			(* Config Cyl ToolTension *)
				ptrTCylToolTension^.T_CtrleCyl.xFBActiv:=TRUE;
				ptrTCylToolTension^.T_Config.xActivState:=TRUE;
				(*22.12.2009: KFS {    *)
				IF xMicroRodActive THEN
				(* Config Cyl ToolLeftActive*)
					ptrTCylToolLeftActive^.T_CtrleCyl.xFBActiv:=TRUE;
					ptrTCylToolLeftActive^.T_Config.xActivState:=TRUE;
				(* Config Cyl ToolRightActive*)
					ptrTCylToolRightActive^.T_CtrleCyl.xFBActiv:=TRUE;
					ptrTCylToolRightActive^.T_Config.xActivState:=TRUE;
				(* Config Cyl ToolCenterActive*)
					ptrTCylToolCenterActive^.T_CtrleCyl.xFBActiv:=TRUE;
					ptrTCylToolCenterActive^.T_Config.xActivState:=TRUE;
				(* Config Cyl ToolPrismaLeftActive*)
					ptrTCylToolPrismaLeftActive^.T_CtrleCyl.xFBActiv:=TRUE;
					ptrTCylToolPrismaLeftActive^.T_Config.xActivState:=TRUE;
				(* Config Cyl ToolPrismaRightActive*)
					ptrTCylToolPrismaRightActive^.T_CtrleCyl.xFBActiv:=TRUE;
					ptrTCylToolPrismaRightActive^.T_Config.xActivState:=TRUE;
				(* Config Cyl ToolWorkLength*)
					ptrTToolFeederWorkLength^.T_CtrleCyl.xFBActiv:=TRUE;
					ptrTToolFeederWorkLength^.T_Config.xActivState:=TRUE;
				END_IF;
				(*22.12.2009: KFS }   *)
			(* Config ToolLeft Axis *)
				ptrTAxisToolLeft^.T_Config_Gen.iTyp:=1;
				ptrTAxisToolLeft^.T_Config_Gen.iMachineType:=iConfigMachineType;
				ptrTAxisToolLeft^.T_Config_ObjFileValue.xSWLimitNeg:=FALSE;
				ptrTAxisToolLeft^.T_Config_ObjFileValue.xSWLimitPos:=FALSE;
				ptrTAxisToolLeft^.T_Config_ObjFileValue.xHWLimitNeg:=FALSE;
				ptrTAxisToolLeft^.T_Config_ObjFileValue.xHWLimitPos:=FALSE;
			(* Config ToolCenter Axis *)
				IF xMicroRodActive THEN
					ptrTAxisToolCenter^.T_Config_Gen.iTyp:=2;
					ptrTAxisToolCenter^.T_Config_Gen.iMachineType:=iConfigMachineType;
					ptrTAxisToolCenter^.T_Config_ObjFileValue.xSWLimitNeg:=FALSE;
					ptrTAxisToolCenter^.T_Config_ObjFileValue.xSWLimitPos:=FALSE;
					ptrTAxisToolCenter^.T_Config_ObjFileValue.xHWLimitNeg:=FALSE;
					ptrTAxisToolCenter^.T_Config_ObjFileValue.xHWLimitPos:=FALSE;
				END_IF;
			(* Config ToolRight Axis *)
				ptrTAxisToolRight^.T_Config_Gen.iTyp:=3;
				ptrTAxisToolRight^.T_Config_Gen.iMachineType:=iConfigMachineType;
				ptrTAxisToolRight^.T_Config_ObjFileValue.xSWLimitNeg:=FALSE;
				ptrTAxisToolRight^.T_Config_ObjFileValue.xSWLimitPos:=FALSE;
				ptrTAxisToolRight^.T_Config_ObjFileValue.xHWLimitNeg:=FALSE;
				ptrTAxisToolRight^.T_Config_ObjFileValue.xHWLimitPos:=FALSE;
			(* Config ToolFeeder Axis *)
				ptrTAxisToolFeeder^.T_Config_Gen.iTyp:=4;
				ptrTAxisToolFeeder^.T_Config_Gen.iMachineType:=iConfigMachineType;
				IF xMicroRodActive THEN
					ptrTAxisToolFeeder^.T_Config_ObjFileValue.xSWLimitNeg:=FALSE;
					ptrTAxisToolFeeder^.T_Config_ObjFileValue.xSWLimitPos:=FALSE;
				   	ptrTAxisToolFeeder^.T_Config_ObjFileValue.xHWLimitNeg:=TRUE;
					ptrTAxisToolFeeder^.T_Config_ObjFileValue.xHWLimitPos:=TRUE;
				ELSE
					ptrTAxisToolFeeder^.T_Config_ObjFileValue.xSWLimitNeg:=FALSE;
					ptrTAxisToolFeeder^.T_Config_ObjFileValue.xSWLimitPos:=FALSE;
					ptrTAxisToolFeeder^.T_Config_ObjFileValue.xHWLimitNeg:=FALSE;
					ptrTAxisToolFeeder^.T_Config_ObjFileValue.xHWLimitPos:=FALSE;
				END_IF;
			(* Config GrindFeeder Axis *)
				ptrTAxisGrindFeeder^.T_Config_Gen.iTyp:=5;
				ptrTAxisGrindFeeder^.T_Config_Gen.iMachineType:=iConfigMachineType;
				ptrTAxisGrindFeeder^.T_Config_ObjFileValue.xSWLimitNeg:=TRUE;
				ptrTAxisGrindFeeder^.T_Config_ObjFileValue.xSWLimitPos:=TRUE;
				ptrTAxisGrindFeeder^.T_Config_ObjFileValue.xHWLimitNeg:=FALSE;
				ptrTAxisGrindFeeder^.T_Config_ObjFileValue.xHWLimitPos:=FALSE;
			END_IF;
			IF NOT(ptrTFunction^.xReset) AND ptrTFunction^.xEnd THEN
				(* Alle Funktionen Resetten *)
				IF (iStationFunctionNr < iMaxFunctionNr) THEN
					iStationFunctionNr:=iStationFunctionNr + 1;
					ptrTFunction^.xReset:=TRUE;
				ELSE
					xInitStep:=FALSE;
					xStartFunction:=FALSE;
					iStepEnable:=200;
				END_IF;
			END_IF;
		110:	IF NOT(xInitStep) THEN
				xInitStep:=TRUE;
				IF TStation.TControl.xHardwareConfigError THEN
					TStation.TControl.xHardwareConfigError:=FALSE;
					TStation.TControl.xActiveHardware:=FALSE;
				ELSE
					xRdyDisableStation:=TRUE;
					xInitStep:=FALSE;
					iStepEnable:=100;
				END_IF;
				RETURN;
			END_IF;
			IF NOT(TStation.TControl.xError) THEN
				TStation.TControl.xActiveHardware:=TRUE;
				xRdyDisableStation:=TRUE;
				xInitStep:=FALSE;
				iStepEnable:=100;
				RETURN;
			END_IF;
		200:	IF NOT(xInitStep) THEN
				xInitStep:=TRUE;
				ptrTCylToolTension^.T_CtrleCyl.xReset:=TRUE;
				(*22.12.2009: KFS {    *)
				IF xMicroRodActive THEN
					ptrTCylToolLeftActive^.T_CtrleCyl.xReset:=TRUE;
					ptrTCylToolRightActive^.T_CtrleCyl.xReset:=TRUE;
					ptrTCylToolCenterActive^.T_CtrleCyl.xReset:=TRUE;
					ptrTCylToolPrismaLeftActive^.T_CtrleCyl.xReset:=TRUE;
					ptrTCylToolPrismaRightActive^.T_CtrleCyl.xReset:=TRUE;
					ptrTToolFeederWorkLength^.T_CtrleCyl.xReset:=TRUE;
				END_IF;
				(*22.12.2009: KFS }   *)
				ptrTAxisToolLeft^.T_CtrleSingle.xReset:=TRUE;
				IF xMicroRodActive THEN
					ptrTAxisToolCenter^.T_CtrleSingle.xReset:=TRUE;
				END_IF;
				ptrTAxisToolRight^.T_CtrleSingle.xReset:=TRUE;
				ptrTAxisToolFeeder^.T_CtrleSingle.xReset:=TRUE;
				ptrTAxisGrindFeeder^.T_CtrleSingle.xReset:=TRUE;
				ptrTAxisGrindSpindle^.T_CtrleSingle.xReset:=TRUE;
			END_IF;
			IF NOT(ptrTAxisToolLeft^.T_CtrleSingle.xReset) AND NOT(ptrTAxisToolCenter^.T_CtrleSingle.xReset) AND ((NOT(ptrTAxisToolRight^.T_CtrleSingle.xReset) AND xMicroRodActive) OR NOT(xMicroRodActive)) AND
			     NOT(ptrTAxisToolFeeder^.T_CtrleSingle.xReset) AND NOT(ptrTAxisGrindFeeder^.T_CtrleSingle.xReset) AND NOT(ptrTAxisGrindSpindle^.T_CtrleSingle.xReset) THEN
				xInitStep:=FALSE;
				IF NOT(xBeckhoffDriveActive) THEN
					iStepEnable:=300;
				ELSE
					iStepEnable:=500;
				END_IF;
			END_IF;
		300:	IF NOT(xInitStep) THEN
				xInitStep:=TRUE;
				ptrTAxisToolLeft^.T_CtrleSingle.lrAcceleration:=T_Standard.T_TeachINToolLeft.rAcceleration;
				ptrTAxisToolLeft^.T_CtrleSingle.lrDecceleration:=T_Standard.T_TeachINToolLeft.rDeceleration;
				ptrTAxisToolCenter^.T_CtrleSingle.lrAcceleration:=T_Standard.T_TeachINToolCenter.rAcceleration;
				ptrTAxisToolCenter^.T_CtrleSingle.lrDecceleration:=T_Standard.T_TeachINToolCenter.rDeceleration;
				ptrTAxisToolRight^.T_CtrleSingle.lrAcceleration:=T_Standard.T_TeachINToolRight.rAcceleration;
				ptrTAxisToolRight^.T_CtrleSingle.lrDecceleration:=T_Standard.T_TeachINToolRight.rDeceleration;
				ptrTAxisToolFeeder^.T_CtrleSingle.lrAcceleration:=T_Standard.T_TeachINToolFeeder.rAcceleration;
				ptrTAxisToolFeeder^.T_CtrleSingle.lrDecceleration:=T_Standard.T_TeachINToolFeeder.rDeceleration;
				ptrTAxisGrindFeeder^.T_CtrleSingle.lrAcceleration:=T_Standard.T_TeachINGrindFeeder.rAcceleration;
				ptrTAxisGrindFeeder^.T_CtrleSingle.lrDecceleration:=T_Standard.T_TeachINGrindFeeder.rDeceleration;
				ptrTAxisToolLeft^.T_Config_Gen.sFileNamePDOMapping:='PDOMapping_ToolLeft';
				ptrTAxisToolLeft^.T_CtrleSingle.iFunction:=22;
				ptrTAxisToolLeft^.T_CtrleSingle.xExecute:=TRUE;
				IF xMicroRodActive THEN
					ptrTAxisToolCenter^.T_Config_Gen.sFileNamePDOMapping:='PDOMapping_ToolCenter';
					ptrTAxisToolCenter^.T_CtrleSingle.iFunction:=22;
					ptrTAxisToolCenter^.T_CtrleSingle.xExecute:=TRUE;
				END_IF;
				ptrTAxisToolRight^.T_Config_Gen.sFileNamePDOMapping:='PDOMapping_ToolRight';
				ptrTAxisToolRight^.T_CtrleSingle.iFunction:=22;
				ptrTAxisToolRight^.T_CtrleSingle.xExecute:=TRUE;
				ptrTAxisToolFeeder^.T_Config_Gen.sFileNamePDOMapping:='PDOMapping_ToolFeeder';
				ptrTAxisToolFeeder^.T_CtrleSingle.iFunction:=22;
				ptrTAxisToolFeeder^.T_CtrleSingle.xExecute:=TRUE;
				ptrTAxisGrindFeeder^.T_Config_Gen.sFileNamePDOMapping:='PDOMapping_GrindFeeder';
				ptrTAxisGrindFeeder^.T_CtrleSingle.iFunction:=22;
				ptrTAxisGrindFeeder^.T_CtrleSingle.xExecute:=TRUE;
				iCountCycle:=0;
			END_IF;
			iCountCycle:=iCountCycle + 1;
			IF (iCountCycle >= 50) THEN
				xReadyChkError:=TRUE;	(* 50 SPS Zyklen warten bis die Übewachung der HW Error freigeschaltet werden kann *)
			END_IF;
			IF xTmp THEN
				RETURN;	(* Wait until all Drives finished *)
			END_IF;
			IF NOT(ptrTAxisToolLeft^.T_CtrleSingle.xExecute) AND ptrTAxisToolLeft^.T_CtrleSingle.xDone AND
			    ((NOT(ptrTAxisToolCenter^.T_CtrleSingle.xExecute) AND ptrTAxisToolCenter^.T_CtrleSingle.xDone AND xMicroRodActive) OR NOT(xMicroRodActive)) AND
			    NOT(ptrTAxisToolRight^.T_CtrleSingle.xExecute) AND ptrTAxisToolRight^.T_CtrleSingle.xDone AND
			    NOT(ptrTAxisToolFeeder^.T_CtrleSingle.xExecute) AND ptrTAxisToolFeeder^.T_CtrleSingle.xDone AND
			    NOT(ptrTAxisGrindFeeder^.T_CtrleSingle.xExecute) AND ptrTAxisGrindFeeder^.T_CtrleSingle.xDone THEN
				xReadyChkError:=TRUE;
				xInitStep:=FALSE;
				iStepEnable:=400;
			END_IF;
		400:	IF NOT(xInitStep) THEN
				xInitStep:=TRUE;
				ptrTAxisToolLeft^.T_CtrleSingle.iFunction:=23;
				ptrTAxisToolLeft^.T_CtrleSingle.xExecute:=TRUE;
				IF xMicroRodActive THEN
					ptrTAxisToolCenter^.T_CtrleSingle.iFunction:=23;
					ptrTAxisToolCenter^.T_CtrleSingle.xExecute:=TRUE;
				END_IF;
				ptrTAxisToolRight^.T_CtrleSingle.iFunction:=23;
				ptrTAxisToolRight^.T_CtrleSingle.xExecute:=TRUE;
				ptrTAxisToolFeeder^.T_CtrleSingle.iFunction:=23;
				ptrTAxisToolFeeder^.T_CtrleSingle.xExecute:=TRUE;
				ptrTAxisGrindFeeder^.T_CtrleSingle.iFunction:=23;
				ptrTAxisGrindFeeder^.T_CtrleSingle.xExecute:=TRUE;
			END_IF;
			IF xTmp THEN
				RETURN;	(* Wait until all Drives finished *)
			END_IF;
			IF NOT(ptrTAxisToolLeft^.T_CtrleSingle.xExecute) AND ptrTAxisToolLeft^.T_CtrleSingle.xDone AND
			    ((NOT(ptrTAxisToolCenter^.T_CtrleSingle.xExecute) AND ptrTAxisToolCenter^.T_CtrleSingle.xDone AND xMicroRodActive) OR NOT(xMicroRodActive)) AND
			    NOT(ptrTAxisToolRight^.T_CtrleSingle.xExecute) AND ptrTAxisToolRight^.T_CtrleSingle.xDone AND
			    NOT(ptrTAxisToolFeeder^.T_CtrleSingle.xExecute) AND ptrTAxisToolFeeder^.T_CtrleSingle.xDone AND
			    NOT(ptrTAxisGrindFeeder^.T_CtrleSingle.xExecute) AND ptrTAxisGrindFeeder^.T_CtrleSingle.xDone THEN
				xInitStep:=FALSE;
				iStepEnable:=500;
			END_IF;
		500:	IF NOT(xInitStep) THEN
				xInitStep:=TRUE;
				ptrTAxisToolLeft^.T_CtrleSingle.iFunction:=1;
				ptrTAxisToolLeft^.T_CtrleSingle.xExecute:=TRUE;
				IF xMicroRodActive THEN
					ptrTAxisToolCenter^.T_CtrleSingle.iFunction:=1;
					ptrTAxisToolCenter^.T_CtrleSingle.xExecute:=TRUE;
				END_IF;
				ptrTAxisToolRight^.T_CtrleSingle.iFunction:=1;
				ptrTAxisToolRight^.T_CtrleSingle.xExecute:=TRUE;
				ptrTAxisToolFeeder^.T_CtrleSingle.iFunction:=1;
				ptrTAxisToolFeeder^.T_CtrleSingle.xExecute:=TRUE;
				ptrTAxisGrindFeeder^.T_CtrleSingle.iFunction:=1;
				ptrTAxisGrindFeeder^.T_CtrleSingle.xExecute:=TRUE;
			END_IF;
			IF NOT(ptrTAxisToolLeft^.T_CtrleSingle.xExecute) AND ptrTAxisToolLeft^.T_CtrleSingle.xDone AND
			    ((NOT(ptrTAxisToolCenter^.T_CtrleSingle.xExecute) AND ptrTAxisToolCenter^.T_CtrleSingle.xDone AND xMicroRodActive) OR NOT(xMicroRodActive)) AND
			    NOT(ptrTAxisToolRight^.T_CtrleSingle.xExecute) AND ptrTAxisToolRight^.T_CtrleSingle.xDone AND
			    NOT(ptrTAxisToolFeeder^.T_CtrleSingle.xExecute) AND ptrTAxisToolFeeder^.T_CtrleSingle.xDone AND
			    NOT(ptrTAxisGrindFeeder^.T_CtrleSingle.xExecute) AND ptrTAxisGrindFeeder^.T_CtrleSingle.xDone THEN
				xInitStep:=FALSE;
				iStepEnable:=600;
			END_IF;
		600:	IF NOT(xInitStep) THEN	(* Read Axis Parameter File *)
				xInitStep:=TRUE;
				ptrTAxisToolLeft^.T_Config_Gen.sDeviceFileName:='EcoStep23S21_ToolLeft';
				ptrTAxisToolLeft^.T_CtrleSingle.iFunction:=2;
				ptrTAxisToolLeft^.T_CtrleSingle.xExecute:=TRUE;
				IF xMicroRodActive THEN
					ptrTAxisToolCenter^.T_Config_Gen.sDeviceFileName:='EcoStep23S21_ToolCenter';
					ptrTAxisToolCenter^.T_CtrleSingle.iFunction:=2;
					ptrTAxisToolCenter^.T_CtrleSingle.xExecute:=TRUE;
				END_IF;
				ptrTAxisToolRight^.T_Config_Gen.sDeviceFileName:='EcoStep23S21_ToolRight';
				ptrTAxisToolRight^.T_CtrleSingle.iFunction:=2;
				ptrTAxisToolRight^.T_CtrleSingle.xExecute:=TRUE;
				ptrTAxisToolFeeder^.T_Config_Gen.sDeviceFileName:='EcoStep23S21_ToolFeeder';
				ptrTAxisToolFeeder^.T_CtrleSingle.iFunction:=2;
				ptrTAxisToolFeeder^.T_CtrleSingle.xExecute:=TRUE;
				ptrTAxisGrindFeeder^.T_Config_Gen.sDeviceFileName:='EcoStep23S21_GrindFeeder';
				ptrTAxisGrindFeeder^.T_CtrleSingle.iFunction:=2;
				ptrTAxisGrindFeeder^.T_CtrleSingle.xExecute:=TRUE;
			END_IF;
			IF NOT(ptrTAxisToolLeft^.T_CtrleSingle.xExecute) AND ptrTAxisToolLeft^.T_CtrleSingle.xDone AND
			    ((NOT(ptrTAxisToolCenter^.T_CtrleSingle.xExecute) AND ptrTAxisToolCenter^.T_CtrleSingle.xDone AND xMicroRodActive) OR NOT(xMicroRodActive)) AND
			    NOT(ptrTAxisToolRight^.T_CtrleSingle.xExecute) AND ptrTAxisToolRight^.T_CtrleSingle.xDone AND
			    NOT(ptrTAxisToolFeeder^.T_CtrleSingle.xExecute) AND ptrTAxisToolFeeder^.T_CtrleSingle.xDone AND
			    NOT(ptrTAxisGrindFeeder^.T_CtrleSingle.xExecute) AND ptrTAxisGrindFeeder^.T_CtrleSingle.xDone THEN
				xInitStep:=FALSE;
				iStepEnable:=700;
			END_IF;
		700:	IF NOT(xInitStep) THEN	(* Read Axis Parameter File *)
				xInitStep:=TRUE;
				ptrTAxisToolLeft^.T_CtrleSingle.iFunction:=21;
				ptrTAxisToolLeft^.T_CtrleSingle.xExecute:=TRUE;
				IF xMicroRodActive THEN
					ptrTAxisToolCenter^.T_CtrleSingle.iFunction:=21;
					ptrTAxisToolCenter^.T_CtrleSingle.xExecute:=TRUE;
				END_IF;
				ptrTAxisToolRight^.T_CtrleSingle.iFunction:=21;
				ptrTAxisToolRight^.T_CtrleSingle.xExecute:=TRUE;
				ptrTAxisToolFeeder^.T_CtrleSingle.iFunction:=21;
				ptrTAxisToolFeeder^.T_CtrleSingle.xExecute:=TRUE;
				ptrTAxisGrindFeeder^.T_CtrleSingle.iFunction:=21;
				ptrTAxisGrindFeeder^.T_CtrleSingle.xExecute:=TRUE;
			END_IF;
			IF NOT(ptrTAxisToolLeft^.T_CtrleSingle.xExecute) AND ptrTAxisToolLeft^.T_CtrleSingle.xDone AND
			    ((NOT(ptrTAxisToolCenter^.T_CtrleSingle.xExecute) AND ptrTAxisToolCenter^.T_CtrleSingle.xDone AND xMicroRodActive) OR NOT(xMicroRodActive)) AND
			    NOT(ptrTAxisToolRight^.T_CtrleSingle.xExecute) AND ptrTAxisToolRight^.T_CtrleSingle.xDone AND
			    NOT(ptrTAxisToolFeeder^.T_CtrleSingle.xExecute) AND ptrTAxisToolFeeder^.T_CtrleSingle.xDone AND
			    NOT(ptrTAxisGrindFeeder^.T_CtrleSingle.xExecute) AND ptrTAxisGrindFeeder^.T_CtrleSingle.xDone THEN
				xInitStep:=FALSE;
				IF NOT(xBeckhoffDriveActive) THEN
					iStepEnable:=1000;
				ELSE
					iStepEnable:=800;
				END_IF;
			END_IF;
		800:	IF NOT(xInitStep) THEN
				IF NOT(T_BoxID.T_Ctrle.xLocked) THEN
					xInitStep:=TRUE;
					(* Box ID-->Beckhoff drive *)
					T_BoxID.T_Ctrle.iMachineType:=iConfigMachineType;
					T_BoxID.T_Servo_ToolLeft.sBoxName:='AX25xx_Slide_St1';
					T_BoxID.T_Servo_ToolLeft.sDeviceName:='AX25xx_Slide_St1';
					T_BoxID.T_Servo_ToolLeft.xDeviceOption:=TRUE;
					T_BoxID.T_Servo_ToolCenter.sBoxName:='AX25xx_Slide_St1';
					T_BoxID.T_Servo_ToolCenter.sDeviceName:='AX25xx_Slide_St1';
					T_BoxID.T_Servo_ToolCenter.xDeviceOption:=TRUE;
					T_BoxID.T_Servo_ToolRight.sBoxName:='AX25xx_Slide_St1';
					T_BoxID.T_Servo_ToolRight.sDeviceName:='AX25xx_Slide_St1';
					T_BoxID.T_Servo_ToolRight.xDeviceOption:=TRUE;
					T_BoxID.T_Servo_ToolFeeder.sBoxName:='AX25xx_Slide_St1';
					T_BoxID.T_Servo_ToolFeeder.sDeviceName:='AX25xx_Slide_St1';
					T_BoxID.T_Servo_ToolFeeder.xDeviceOption:=TRUE;
					T_BoxID.T_Servo_GrindFeeder.sBoxName:='AX25xx_Slide_St1';
					T_BoxID.T_Servo_GrindFeeder.sDeviceName:='AX25xx_Slide_St1';
					T_BoxID.T_Servo_GrindFeeder.xDeviceOption:=TRUE;
					T_BoxID.T_Ctrle.xLocked:=TRUE;
					T_BoxID.T_Ctrle.xExecute:=TRUE;
				END_IF;
				RETURN;
			END_IF;
			IF NOT(T_BoxID.T_Ctrle.xExecute) AND T_BoxID.T_Ctrle.xDone AND T_BoxID.T_Ctrle.xLocked THEN
				T_BoxID.T_Ctrle.xLocked:=FALSE;
				xInitStep:=FALSE;
				iStepEnable:=900;
			END_IF;
		900:	IF NOT(xInitStep) THEN
				xInitStep:=TRUE;
				IF (T_BoxID.T_Servo_ToolLeft.wAddrBox = 0) OR (T_BoxID.T_Servo_ToolLeft.wAddrBox <> ptrTAxisToolLeft^.T_Config_Gen.udiNC_TaskIdxGrp) THEN
					xSetError:=TRUE;
					diErrorNumber:=16#F201;	(* ToolLeft-->Falsche Konfiguration oder Achse nicht vorhanden *)
					RETURN;
				ELSIF ((T_BoxID.T_Servo_ToolCenter.wAddrBox = 0) OR (T_BoxID.T_Servo_ToolCenter.wAddrBox <> ptrTAxisToolCenter^.T_Config_Gen.udiNC_TaskIdxGrp)) AND xMicroRodActive THEN
					xSetError:=TRUE;
					diErrorNumber:=16#F202;	(* ToolCenter-->Falsche Konfiguration oder Achse nicht vorhanden *)
					RETURN;
				ELSIF (T_BoxID.T_Servo_ToolRight.wAddrBox = 0) OR (T_BoxID.T_Servo_ToolRight.wAddrBox <> ptrTAxisToolRight^.T_Config_Gen.udiNC_TaskIdxGrp) THEN
					xSetError:=TRUE;
					diErrorNumber:=16#F203;	(* ToolRight-->Falsche Konfiguration oder Achse nicht vorhanden *)
					RETURN;
				ELSIF (T_BoxID.T_Servo_ToolFeeder.wAddrBox = 0) OR (T_BoxID.T_Servo_ToolFeeder.wAddrBox <> ptrTAxisToolFeeder^.T_Config_Gen.udiNC_TaskIdxGrp) THEN
					xSetError:=TRUE;
					diErrorNumber:=16#F204;	(* ToolFeeder-->Falsche Konfiguration oder Achse nicht vorhanden *)
					RETURN;
				ELSIF (T_BoxID.T_Servo_GrindFeeder.wAddrBox = 0) OR (T_BoxID.T_Servo_GrindFeeder.wAddrBox <> ptrTAxisGrindFeeder^.T_Config_Gen.udiNC_TaskIdxGrp) THEN
					xSetError:=TRUE;
					diErrorNumber:=16#F205;	(* GrindFeeder-->Falsche Konfiguration oder Achse nicht vorhanden *)
					RETURN;
				ELSE
				(* Achsenparameterisierung erfolgreich *)
					;
				END_IF;
				xInitStep:=FALSE;
				iStepEnable:=1100;
			END_IF;
		(* Read Axis Firmware Information *)
		1000:IF NOT(xInitStep) THEN
				xInitStep:=TRUE;
				ptrTAxisToolLeft^.T_CtrleSingle.iFunction:=27;
				ptrTAxisToolLeft^.T_CtrleSingle.xExecute:=TRUE;
				IF xMicroRodActive THEN
					ptrTAxisToolCenter^.T_CtrleSingle.iFunction:=27;
					ptrTAxisToolCenter^.T_CtrleSingle.xExecute:=TRUE;
				END_IF;
				ptrTAxisToolRight^.T_CtrleSingle.iFunction:=27;
				ptrTAxisToolRight^.T_CtrleSingle.xExecute:=TRUE;
				ptrTAxisToolFeeder^.T_CtrleSingle.iFunction:=27;
				ptrTAxisToolFeeder^.T_CtrleSingle.xExecute:=TRUE;
				ptrTAxisGrindFeeder^.T_CtrleSingle.iFunction:=27;
				ptrTAxisGrindFeeder^.T_CtrleSingle.xExecute:=TRUE;
			END_IF;
			IF NOT(ptrTAxisToolLeft^.T_CtrleSingle.xExecute) AND ptrTAxisToolLeft^.T_CtrleSingle.xDone AND
			    ((NOT(ptrTAxisToolCenter^.T_CtrleSingle.xExecute) AND ptrTAxisToolCenter^.T_CtrleSingle.xDone AND xMicroRodActive) OR NOT(xMicroRodActive)) AND
			    NOT(ptrTAxisToolRight^.T_CtrleSingle.xExecute) AND ptrTAxisToolRight^.T_CtrleSingle.xDone AND
			    NOT(ptrTAxisToolFeeder^.T_CtrleSingle.xExecute) AND ptrTAxisToolFeeder^.T_CtrleSingle.xDone AND
			    NOT(ptrTAxisGrindFeeder^.T_CtrleSingle.xExecute) AND ptrTAxisGrindFeeder^.T_CtrleSingle.xDone THEN
				xInitStep:=FALSE;
				iStepEnable:=1100;
			END_IF;
		1100:IF NOT(xInitStep) THEN
				xInitStep:=TRUE;
				ptrTAxisToolLeft^.T_CtrleSingle.iFunction:=4;
				ptrTAxisToolLeft^.T_CtrleSingle.xExecute:=TRUE;
				IF xMicroRodActive THEN
					ptrTAxisToolCenter^.T_CtrleSingle.iFunction:=4;
					ptrTAxisToolCenter^.T_CtrleSingle.xExecute:=TRUE;
				END_IF;
				ptrTAxisToolRight^.T_CtrleSingle.iFunction:=4;
				ptrTAxisToolRight^.T_CtrleSingle.xExecute:=TRUE;
				ptrTAxisToolFeeder^.T_CtrleSingle.iFunction:=4;
				ptrTAxisToolFeeder^.T_CtrleSingle.xExecute:=TRUE;
				ptrTAxisGrindFeeder^.T_CtrleSingle.iFunction:=4;
				ptrTAxisGrindFeeder^.T_CtrleSingle.xExecute:=TRUE;
				ptrTAxisGrindSpindle^.T_CtrleSingle.iFunction:=4;
				ptrTAxisGrindSpindle^.T_CtrleSingle.xExecute:=TRUE;
			END_IF;
			IF NOT(ptrTAxisToolLeft^.T_CtrleSingle.xExecute) AND ptrTAxisToolLeft^.T_CtrleSingle.xDone AND
			    ((NOT(ptrTAxisToolCenter^.T_CtrleSingle.xExecute) AND ptrTAxisToolCenter^.T_CtrleSingle.xDone AND xMicroRodActive) OR NOT(xMicroRodActive)) AND
			    NOT(ptrTAxisToolRight^.T_CtrleSingle.xExecute) AND ptrTAxisToolRight^.T_CtrleSingle.xDone AND
			    NOT(ptrTAxisToolFeeder^.T_CtrleSingle.xExecute) AND ptrTAxisToolFeeder^.T_CtrleSingle.xDone AND
			    NOT(ptrTAxisGrindFeeder^.T_CtrleSingle.xExecute) AND ptrTAxisGrindFeeder^.T_CtrleSingle.xDone AND
			    NOT(ptrTAxisGrindSpindle^.T_CtrleSingle.xExecute) AND ptrTAxisGrindSpindle^.T_CtrleSingle.xDone THEN
				xInitStep:=FALSE;
				iStepEnable:=1200;
			END_IF;
		1200:IF NOT(xInitStep) THEN
				xInitStep:=TRUE;
				ptrTAxisToolLeft^.T_CtrleSingle.iFunction:=3;
				ptrTAxisToolLeft^.T_CtrleSingle.xExecute:=TRUE;
				IF xMicroRodActive THEN
					ptrTAxisToolCenter^.T_CtrleSingle.iFunction:=3;
					ptrTAxisToolCenter^.T_CtrleSingle.xExecute:=TRUE;
				END_IF;
				ptrTAxisToolRight^.T_CtrleSingle.iFunction:=3;
				ptrTAxisToolRight^.T_CtrleSingle.xExecute:=TRUE;
				ptrTAxisToolFeeder^.T_CtrleSingle.iFunction:=3;
				ptrTAxisToolFeeder^.T_CtrleSingle.xExecute:=TRUE;
				ptrTAxisGrindFeeder^.T_CtrleSingle.iFunction:=3;
				ptrTAxisGrindFeeder^.T_CtrleSingle.xExecute:=TRUE;
			END_IF;
			IF NOT(ptrTAxisToolLeft^.T_CtrleSingle.xExecute) AND ptrTAxisToolLeft^.T_CtrleSingle.xDone AND
			    ((NOT(ptrTAxisToolCenter^.T_CtrleSingle.xExecute) AND ptrTAxisToolCenter^.T_CtrleSingle.xDone AND xMicroRodActive) OR NOT(xMicroRodActive)) AND
			    NOT(ptrTAxisToolRight^.T_CtrleSingle.xExecute) AND ptrTAxisToolRight^.T_CtrleSingle.xDone AND
			    NOT(ptrTAxisToolFeeder^.T_CtrleSingle.xExecute) AND ptrTAxisToolFeeder^.T_CtrleSingle.xDone AND
			    NOT(ptrTAxisGrindFeeder^.T_CtrleSingle.xExecute) AND ptrTAxisGrindFeeder^.T_CtrleSingle.xDone THEN
				IF NOT(xFirstTimeBooting) THEN
					xFirstTimeBooting:=TRUE;
					iStepEnable:=1300;
				ELSE
					iStepEnable:=1400;
				END_IF;
				xInitStep:=FALSE;
			END_IF;
		(* Set the Position of the GrindFeeder on the Settled ToolDiameter, but only on the first time on booting of the machine *)
		1300:IF NOT(xInitStep) THEN
				xInitStep:=TRUE;
				ptrTAxisGrindFeeder^.T_CtrleSingle.rSetPosition:=T_ProcessImageData.T_ProcessPara.rToolDiameterProcess;
				ptrTAxisGrindFeeder^.T_CtrleSingle.iFunction:=11;
				ptrTAxisGrindFeeder^.T_CtrleSingle.xExecute:=TRUE;
			END_IF;
			IF NOT(ptrTAxisGrindFeeder^.T_CtrleSingle.xExecute) AND ptrTAxisGrindFeeder^.T_CtrleSingle.xDone THEN
				xInitStep:=FALSE;
				iStepEnable:=1400;
			END_IF;
		(* Set the SW Limit position for the GrindFeeder Axis *)
		1400:IF NOT(xInitStep) THEN
				xInitStep:=TRUE;
				ptrTAxisGrindFeeder^.T_CtrleSingle.lrSWNegLimitSwitch:=T_ProcessImageData.T_PrismPara.rToolDiameterMin;
				ptrTAxisGrindFeeder^.T_CtrleSingle.lrSWPosLimitSwitch:=T_ProcessImageData.T_PrismPara.rToolDiameterMax + T_Standard.T_TeachINGrindFeeder.rOffsetSWPosEndSwitch;
				ptrTAxisGrindFeeder^.T_CtrleSingle.iFunction:=28;
				ptrTAxisGrindFeeder^.T_CtrleSingle.xExecute:=TRUE;
			END_IF;
			IF NOT(ptrTAxisGrindFeeder^.T_CtrleSingle.xExecute) AND ptrTAxisGrindFeeder^.T_CtrleSingle.xDone THEN
				xInitStep:=FALSE;
				IF NOT(xMicroRodActive) THEN
					(* Only for MicroWire activate the ToolTension *)
					iStepEnable:=1500;
				ELSE
					iStepEnable:=1600;
				END_IF;
			END_IF;
		1500:IF NOT(xInitStep) THEN
				xInitStep:=TRUE;
				ptrTCylToolTension^.T_CtrleCyl.iFunction:=2;
				ptrTCylToolTension^.T_CtrleCyl.T_AnalogCylinder.rForceIn:=T_ProcessImageData.T_ProcessPara.rToolTensionProcess;
				ptrTCylToolTension^.T_CtrleCyl.xExecute:=TRUE;
			END_IF;
			IF NOT(ptrTCylToolTension^.T_CtrleCyl.xExecute) AND ptrTCylToolTension^.T_CtrleCyl.xDone THEN
				xInitStep:=FALSE;
				iStepEnable:=1600;
			END_IF;
		1600:xReadyChkError:=FALSE;
			xInitStep:=FALSE;
			xSetEnableConfig:=TRUE;
			iEnableConfigMachineType:=iConfigMachineType;
			iEnableConfigAxisType:=iConfigAxisType;
			iEnableConfigVisuNavigation:=iConfigVisuNavigation;
			rEnableConfigMaxToolLength:=rConfigMaxToolLength;
			xInitSetEnable:=FALSE;
			TStation.TControl.xRdy:=TRUE;
			xSetEnd:=TRUE;
	END_CASE;
END_IF;
END_ACTION
ACTION CtrlErrorStation:
IF xStationError OR xForceHWError OR (ptrTFunction^.xError AND TStation.TControl.xRdy AND NOT(xSetEnd)) THEN
	IF NOT(xInitError) THEN
		xForceHWError:=FALSE;
		xStationError:=TRUE;
		xTmpStationError:=TRUE;
		xInitError:=TRUE;
		xAxisErrorActive:=FALSE;
		TStation.TControl.diErrorNr:=0;
		IF ptrTAxisToolLeft^.T_CtrleSingle.xErr THEN
			TStation.TControl.diErrorNr:=1000000 + ptrTAxisToolLeft^.T_CtrleSingle.udiErrorID;
			ptrTAxisToolLeft^.T_CtrleSingle.iFunction:=1;
			ptrTAxisToolLeft^.T_CtrleSingle.xExecute:=TRUE;
			xAxisErrorActive:=TRUE;
		END_IF;
		IF xMicroRodActive THEN
			IF ptrTAxisToolCenter^.T_CtrleSingle.xErr THEN
				TStation.TControl.diErrorNr:=2000000 + ptrTAxisToolCenter^.T_CtrleSingle.udiErrorID;
				ptrTAxisToolCenter^.T_CtrleSingle.iFunction:=1;
				ptrTAxisToolCenter^.T_CtrleSingle.xExecute:=TRUE;
				xAxisErrorActive:=TRUE;
			END_IF;
		END_IF;
		IF ptrTAxisToolRight^.T_CtrleSingle.xErr THEN
			TStation.TControl.diErrorNr:=3000000 + ptrTAxisToolRight^.T_CtrleSingle.udiErrorID;
			ptrTAxisToolRight^.T_CtrleSingle.iFunction:=1;
			ptrTAxisToolRight^.T_CtrleSingle.xExecute:=TRUE;
			xAxisErrorActive:=TRUE;
		END_IF;
		IF ptrTAxisToolFeeder^.T_CtrleSingle.xErr THEN
			TStation.TControl.diErrorNr:=4000000 + ptrTAxisToolFeeder^.T_CtrleSingle.udiErrorID;
			ptrTAxisToolFeeder^.T_CtrleSingle.iFunction:=1;
			ptrTAxisToolFeeder^.T_CtrleSingle.xExecute:=TRUE;
			xAxisErrorActive:=TRUE;
		END_IF;
		IF ptrTAxisGrindFeeder^.T_CtrleSingle.xErr THEN
			TStation.TControl.diErrorNr:=5000000 + ptrTAxisGrindFeeder^.T_CtrleSingle.udiErrorID;
			ptrTAxisGrindFeeder^.T_CtrleSingle.iFunction:=1;
			ptrTAxisGrindFeeder^.T_CtrleSingle.xExecute:=TRUE;
			xAxisErrorActive:=TRUE;
		END_IF;
		IF ptrTCylToolTension^.T_CtrleCyl.xErr THEN
			TStation.TControl.diErrorNr:=6000000 + ptrTCylToolTension^.T_CtrleCyl.udiErrorID;
			ptrTCylToolTension^.T_CtrleCyl.xReset:=TRUE;
		END_IF;
		IF (TStation.TControl.diErrorNr = 0) THEN	(* General Error-->No Hardware Error  7000 - 7999*)
			TStation.TControl.diErrorNr:=8000000 + ptrTFunction^.iErrorNr;
		END_IF;
		ptrTFunction^.xQuitErr:=NOT(ptrTFunction^.xEnd) AND ptrTFunction^.xError;
		IF NOT(ptrTFunction^.xQuitErr) AND NOT(ptrTFunction^.xEnd) THEN
			xForceResetAxis:=TRUE;
			ptrTFunction^.xReset:=TRUE;
		END_IF;
		TONWaitReset(IN:=FALSE);
	END_IF;
	IF (ptrTFunction^.xEnd OR xForceResetAxis) AND xTmpStationError THEN
		IF NOT(ptrTAxisToolLeft^.T_CtrleSingle.xErr) AND ((NOT(ptrTAxisToolCenter^.T_CtrleSingle.xErr) AND xMicroRodActive) OR NOT(xMicroRodActive)) AND
		     NOT(ptrTAxisToolRight^.T_CtrleSingle.xErr) AND NOT(ptrTAxisToolFeeder^.T_CtrleSingle.xErr) AND NOT(ptrTAxisGrindFeeder^.T_CtrleSingle.xErr) THEN
			TStation.TControl.xError:=TRUE;
			xForceResetAxis:=FALSE;
		END_IF;
		TONWaitReset(IN:=TRUE,PT:=T#100ms);
		IF TONWaitReset.Q THEN
			IF xAxisErrorActive THEN
				T_StartUp.T_Ctrle.xSetSecurityStateON:=TRUE;
			END_IF;
			xStepError:=FALSE;
			xStartFunction:=FALSE;
			xTmpStationError:=FALSE;
			xReadyToQuitErr:=TRUE;
		END_IF;
	END_IF;
	IF TStation.TControl.xQuitError AND NOT(ptrTFunction^.xQuitErr) AND xReadyToQuitErr THEN
		xInitError:=FALSE;
		TStation.TControl.xQuitError:=FALSE;
		xSetEnd:=TRUE;
	END_IF;
END_IF;
END_ACTION
ACTION CtrlMainStation:
IF (TStation.TControl.xStart OR xTmpStart) AND TStation.TControl.xRdy AND NOT(xSetEnd) THEN
	IF NOT(xInitStart) THEN
		xInitStart:=TRUE;
		xTmpStart:=TRUE;
		TStation.TControl.xStart:=FALSE;
		TStation.TControl.xEnd:=FALSE;
		ptrTFunction^.xStart:=TRUE;
		xStartFunction:=TRUE;
		iStationFunctionNr:=TStation.TControl.iFunctNr;
		TStation.TControl.xAbord:=FALSE;
	END_IF;
	IF TStation.TControl.xStop THEN
		IF NOT(xInitStop) THEN
			xInitStop:=TRUE;
			ptrTFunction^.xStop:=TRUE;
		END_IF;
		IF NOT(ptrTFunction^.xStop) THEN
			xInitStop:=FALSE;
			TStation.TControl.xStop:=FALSE;
			xTmpStopFunction:=TRUE;
		END_IF;
	END_IF;
	IF TStation.TControl.xStart AND xTmpStopFunction AND NOT(ptrTFunction^.xAbord) THEN
		TStation.TControl.xStart:=FALSE;
		xTmpStopFunction:=FALSE;
		ptrTFunction^.xStart:=TRUE;
	END_IF;
	IF TStation.TControl.xAbord AND xTmpStopFunction THEN
		TStation.TControl.xAbord:=FALSE;
		xTmpStopFunction:=FALSE;
		ptrTFunction^.xStart:=FALSE;
		ptrTFunction^.xAbord:=TRUE;
	END_IF;
	IF NOT(ptrTFunction^.xStart) AND ptrTFunction^.xEnd AND NOT(xStationError) THEN
		xTmpStart:=FALSE;
		xInitStart:=FALSE;
		xSetEnd:=TRUE;
	END_IF;
END_IF;
END_ACTION
ACTION CtrlSafetySwitch_ON_OFF:
(******************************************************************************************************************************************)
(****************************				       Security Circuit Switch ON/OFF                                          *****************************)
(******************************************************************************************************************************************)
IF (TStation.TControl.xSecurityCircuitOn OR TStation.TControl.xSecurityCircuitOff OR xSecurityCircuitOn OR xSecurityCircuitOff) AND NOT(xInitSetEnable) AND NOT(xInitDelEnable) THEN
	IF NOT(xSecurityCircuitOn) AND NOT(xSecurityCircuitOff) THEN
		xSecurityCircuitOn:=TStation.TControl.xSecurityCircuitOn;
		xSecurityCircuitOff:=TStation.TControl.xSecurityCircuitOff;
		iStepSecCircuit:=1;
		xInitSecCircuit:=FALSE;
		TStation.TControl.xRdy:=FALSE;
		TStation.TControl.xEnd:=FALSE;
		TONCheckTimeOut(IN:=FALSE);
	END_IF;
	IF xSecurityCircuitOn THEN
		IF TStation.TControl.xSecurityCircuitOff THEN
			TStation.TControl.xSecurityCircuitOn:=FALSE;
			xSecurityCircuitOn:=FALSE;
		END_IF;
	END_IF;
	IF xSecurityCircuitOff THEN
		IF TStation.TControl.xSecurityCircuitOn THEN
			TStation.TControl.xSecurityCircuitOff:=FALSE;
			xSecurityCircuitOff:=FALSE;
		END_IF;
	END_IF;
	TONCheckTimeOut(IN:=TRUE,PT:=T#0.5s);
	xCheckAxisError:=FALSE;
	IF TONCheckTimeOut.Q THEN
		IF ptrTAxisToolLeft^.T_CtrleSingle.xErr THEN
			ptrTAxisToolLeft^.T_CtrleSingle.iFunction:=1;
			ptrTAxisToolLeft^.T_CtrleSingle.xExecute:=TRUE;
			xCheckAxisError:=TRUE;
		END_IF;
		IF xMicroRodActive THEN
			IF ptrTAxisToolCenter^.T_CtrleSingle.xErr THEN
				ptrTAxisToolCenter^.T_CtrleSingle.iFunction:=1;
				ptrTAxisToolCenter^.T_CtrleSingle.xExecute:=TRUE;
				xCheckAxisError:=TRUE;
			END_IF;
		END_IF;
		IF ptrTAxisToolRight^.T_CtrleSingle.xErr THEN
			ptrTAxisToolRight^.T_CtrleSingle.iFunction:=1;
			ptrTAxisToolRight^.T_CtrleSingle.xExecute:=TRUE;
			xCheckAxisError:=TRUE;
		END_IF;
		IF ptrTAxisToolFeeder^.T_CtrleSingle.xErr THEN
			ptrTAxisToolFeeder^.T_CtrleSingle.iFunction:=1;
			ptrTAxisToolFeeder^.T_CtrleSingle.xExecute:=TRUE;
			xCheckAxisError:=TRUE;
		END_IF;
		IF ptrTAxisGrindFeeder^.T_CtrleSingle.xErr THEN
			ptrTAxisGrindFeeder^.T_CtrleSingle.iFunction:=1;
			ptrTAxisGrindFeeder^.T_CtrleSingle.xExecute:=TRUE;
			xCheckAxisError:=TRUE;
		END_IF;
		TStation.TControl.xRdy:=TRUE;
		IF xCheckAxisError THEN
			TStation.TControl.xSecurityCircuitOn:=FALSE;
			TStation.TControl.xSecurityCircuitOff:=FALSE;
			xSecurityCircuitOn:=FALSE;
			xSecurityCircuitOff:=FALSE;
			iStepSecCircuit:=1;
			xInitSecCircuit:=FALSE;
			xSetEnd:=TRUE;
			RETURN;
		END_IF;
	END_IF;
	CASE iStepSecCircuit OF
	1:	IF NOT(xInitSecCircuit) THEN
			xInitSecCircuit:=TRUE;
			ptrTFunction^.xReset:=TRUE;
			iStationFunctionNr:=1;
			xStartFunction:=TRUE;
		END_IF;
		IF NOT(ptrTFunction^.xReset) AND ptrTFunction^.xEnd THEN
			(* Alle Funktionen Resetten *)
			IF (iStationFunctionNr < iMaxFunctionNr) THEN
				iStationFunctionNr:=iStationFunctionNr + 1;
				ptrTFunction^.xReset:=TRUE;
			ELSE
				xInitSecCircuit:=FALSE;
				iStepSecCircuit:=10;
				xStartFunction:=FALSE;
			END_IF;
		END_IF;
	10:	IF NOT(xInitSecCircuit) THEN
			xInitSecCircuit:=TRUE;
			ptrTAxisToolLeft^.T_CtrleSingle.xReset:=TRUE;
			IF xMicroRodActive THEN
				ptrTAxisToolCenter^.T_CtrleSingle.xReset:=TRUE;
			END_IF;
			ptrTAxisToolRight^.T_CtrleSingle.xReset:=TRUE;
			ptrTAxisToolFeeder^.T_CtrleSingle.xReset:=TRUE;
			ptrTAxisGrindFeeder^.T_CtrleSingle.xReset:=TRUE;
			ptrTAxisGrindSpindle^.T_CtrleSingle.xReset:=TRUE;
		END_IF;
		IF NOT(ptrTAxisToolLeft^.T_CtrleSingle.xReset) AND ((NOT(ptrTAxisToolCenter^.T_CtrleSingle.xReset) AND xMicroRodActive) OR NOT(xMicroRodActive)) AND NOT(ptrTAxisToolRight^.T_CtrleSingle.xReset) AND
		    NOT(ptrTAxisToolFeeder^.T_CtrleSingle.xReset) AND NOT(ptrTAxisGrindFeeder^.T_CtrleSingle.xReset) AND NOT(ptrTAxisGrindSpindle^.T_CtrleSingle.xReset) THEN
			xInitSecCircuit:=FALSE;
			iStepSecCircuit:=20;
		END_IF;
	20:	IF NOT(xInitSecCircuit) THEN
			xInitSecCircuit:=TRUE;
			ptrTAxisToolLeft^.T_CtrleSingle.iFunction:=1;
			ptrTAxisToolLeft^.T_CtrleSingle.xExecute:=TRUE;
			IF xMicroRodActive THEN
				ptrTAxisToolCenter^.T_CtrleSingle.iFunction:=1;
				ptrTAxisToolCenter^.T_CtrleSingle.xExecute:=TRUE;
			END_IF;
			ptrTAxisToolRight^.T_CtrleSingle.iFunction:=1;
			ptrTAxisToolRight^.T_CtrleSingle.xExecute:=TRUE;
			ptrTAxisToolFeeder^.T_CtrleSingle.iFunction:=1;
			ptrTAxisToolFeeder^.T_CtrleSingle.xExecute:=TRUE;
			ptrTAxisGrindFeeder^.T_CtrleSingle.iFunction:=1;
			ptrTAxisGrindFeeder^.T_CtrleSingle.xExecute:=TRUE;
			ptrTAxisGrindSpindle^.T_CtrleSingle.iFunction:=1;
			ptrTAxisGrindSpindle^.T_CtrleSingle.xExecute:=TRUE;
		END_IF;
		IF NOT(ptrTAxisToolLeft^.T_CtrleSingle.xExecute) AND ptrTAxisToolLeft^.T_CtrleSingle.xDone AND
		    ((NOT(ptrTAxisToolCenter^.T_CtrleSingle.xExecute) AND ptrTAxisToolCenter^.T_CtrleSingle.xDone AND xMicroRodActive) OR NOT(xMicroRodActive)) AND
		    NOT(ptrTAxisToolRight^.T_CtrleSingle.xExecute) AND ptrTAxisToolRight^.T_CtrleSingle.xDone AND
		    NOT(ptrTAxisToolFeeder^.T_CtrleSingle.xExecute) AND ptrTAxisToolFeeder^.T_CtrleSingle.xDone AND
		    NOT(ptrTAxisGrindFeeder^.T_CtrleSingle.xExecute) AND ptrTAxisGrindFeeder^.T_CtrleSingle.xDone AND
		    NOT(ptrTAxisGrindSpindle^.T_CtrleSingle.xExecute) AND ptrTAxisGrindSpindle^.T_CtrleSingle.xDone THEN
			xInitSecCircuit:=FALSE;
			iStepSecCircuit:=30;
		END_IF;
	30:	IF NOT(xInitSecCircuit) THEN
			xInitSecCircuit:=TRUE;
			(* Resetten der Aktuatoren *)
			ptrTCylToolTension^.T_CtrleCyl.xReset:=TRUE;
			(*22.12.2009: KFS {    *)
			IF xMicroRodActive THEN
				ptrTCylToolLeftActive^.T_CtrleCyl.xReset:=TRUE;
				ptrTCylToolRightActive^.T_CtrleCyl.xReset:=TRUE;
				ptrTCylToolCenterActive^.T_CtrleCyl.xReset:=TRUE;
				ptrTCylToolPrismaLeftActive^.T_CtrleCyl.xReset:=TRUE;
				ptrTCylToolPrismaRightActive^.T_CtrleCyl.xReset:=TRUE;
			END_IF;
			(*22.12.2009: KFS }   *)
		END_IF;
		IF NOT(ptrTCylToolTension^.T_CtrleCyl.xReset) AND ptrTCylToolTension^.T_CtrleCyl.xDone AND
		     ( NOT(xMicroRodActive) OR
		         ( NOT(ptrTCylToolLeftActive^.T_CtrleCyl.xReset) AND ptrTCylToolLeftActive^.T_CtrleCyl.xDone AND
		           NOT(ptrTCylToolRightActive^.T_CtrleCyl.xReset) AND ptrTCylToolRightActive^.T_CtrleCyl.xDone AND
		           NOT(ptrTCylToolCenterActive^.T_CtrleCyl.xReset) AND ptrTCylToolCenterActive^.T_CtrleCyl.xDone AND
 		           NOT(ptrTCylToolPrismaLeftActive^.T_CtrleCyl.xReset) AND ptrTCylToolPrismaLeftActive^.T_CtrleCyl.xDone AND
                              NOT(ptrTCylToolPrismaRightActive^.T_CtrleCyl.xReset) AND ptrTCylToolPrismaRightActive^.T_CtrleCyl.xDone )  )  THEN
			xInitSecCircuit:=FALSE;
			IF xSecurityCircuitOn THEN
				iStepSecCircuit:=40;
			ELSE
				iStepSecCircuit:=50;
			END_IF;
		END_IF;
	40:	IF NOT(xInitSecCircuit) THEN
				xInitSecCircuit:=TRUE;
				ptrTAxisToolLeft^.T_CtrleSingle.iFunction:=3;
				ptrTAxisToolLeft^.T_CtrleSingle.xExecute:=TRUE;
				IF xMicroRodActive THEN
					ptrTAxisToolCenter^.T_CtrleSingle.iFunction:=3;
					ptrTAxisToolCenter^.T_CtrleSingle.xExecute:=TRUE;
				END_IF;
				ptrTAxisToolRight^.T_CtrleSingle.iFunction:=3;
				ptrTAxisToolRight^.T_CtrleSingle.xExecute:=TRUE;
				ptrTAxisToolFeeder^.T_CtrleSingle.iFunction:=3;
				ptrTAxisToolFeeder^.T_CtrleSingle.xExecute:=TRUE;
				ptrTAxisGrindFeeder^.T_CtrleSingle.iFunction:=3;
				ptrTAxisGrindFeeder^.T_CtrleSingle.xExecute:=TRUE;
				IF NOT(xMicroRodActive) THEN
					ptrTCylToolTension^.T_CtrleCyl.iFunction:=2;
					IF (iSelectToolTensionForce < 2) THEN
						ptrTCylToolTension^.T_CtrleCyl.T_AnalogCylinder.rForceIn:=T_ProcessImageData.T_ProcessPara.rToolTensionProcess;
					END_IF;
					IF (iSelectToolTensionForce > 1) THEN
						ptrTCylToolTension^.T_CtrleCyl.T_AnalogCylinder.rForceIn:=T_Standard.T_Cyl_ToolTension.rForce;
					END_IF
					ptrTCylToolTension^.T_CtrleCyl.xExecute:=TRUE;
				END_IF;
			END_IF;
			IF NOT(ptrTAxisToolLeft^.T_CtrleSingle.xExecute) AND ptrTAxisToolLeft^.T_CtrleSingle.xDone AND
			    ((NOT(ptrTAxisToolCenter^.T_CtrleSingle.xExecute) AND ptrTAxisToolCenter^.T_CtrleSingle.xDone AND xMicroRodActive) OR NOT(xMicroRodActive)) AND
			    NOT(ptrTAxisToolRight^.T_CtrleSingle.xExecute) AND ptrTAxisToolRight^.T_CtrleSingle.xDone AND
			    NOT(ptrTAxisToolFeeder^.T_CtrleSingle.xExecute) AND ptrTAxisToolFeeder^.T_CtrleSingle.xDone AND
			    NOT(ptrTAxisGrindFeeder^.T_CtrleSingle.xExecute) AND ptrTAxisGrindFeeder^.T_CtrleSingle.xDone AND
			    ((NOT(ptrTCylToolTension^.T_CtrleCyl.xExecute) AND ptrTCylToolTension^.T_CtrleCyl.xDone AND NOT(xMicroRodActive)) OR xMicroRodActive) THEN
				xInitSecCircuit:=FALSE;
				iStepSecCircuit:=50;
			END_IF;
	50:	TStation.TControl.xRdy:=TRUE;
		TStation.TControl.xSecurityCircuitOn:=FALSE;
		TStation.TControl.xSecurityCircuitOff:=FALSE;
		xSecurityCircuitOn:=FALSE;
		xSecurityCircuitOff:=FALSE;
		iStepSecCircuit:=1;
		xInitSecCircuit:=FALSE;
		xSetEnd:=TRUE;
	END_CASE;
ELSE
	TStation.TControl.xSecurityCircuitOn:=FALSE;
	TStation.TControl.xSecurityCircuitOff:=FALSE;
	xSecurityCircuitOn:=FALSE;
	xSecurityCircuitOff:=FALSE;
	iStepSecCircuit:=1;
	xInitSecCircuit:=FALSE;
	TONCheckTimeOut(IN:=FALSE);
END_IF;
END_ACTION

(* POU PRG_STATION_LAYER3/FB_STATIONEN/FB_FUNCTION/FB_FctToolRotationTorqueStart, ST *)
FUNCTION_BLOCK FB_FctToolRotationTorqueStart
VAR_INPUT
	xMicroRodActive: BOOL;		(* choice of the machine MicroWire or MicroRod *)
	xBeckhoffDriveActive: BOOL;	(* choice of the axis Beckhoff or EcoStep *)
	xSafetyCircuitOn:BOOL;			(* state of the safety circuit-->TRUE=Machine current ON, FALSE=Machine current OFF *)
END_VAR
VAR_IN_OUT
	xStart : BOOL;					(* start the function *)
	xReset : BOOL;				(* reset the function *)
	xStop : BOOL;					(* stop the active function *)
	xQuitErr : BOOL;				(* quit the error caused of the active function *)
	xAbord : BOOL;				(* abord the active function *)
	TAxisToolLeft:ST_AXIS;		(* data structure for the ToolLeft axis *)
	TAxisToolCenter:ST_AXIS;		(* data structure for the ToolCenter axis *)
	TAxisToolRight:ST_AXIS;		(* data structure for the ToolRight axis *)
	TAxisToolFeeder:ST_AXIS;		(* data structure for the ToolFeeder axis *)
END_VAR
VAR_OUTPUT
	xEnd : BOOL;					(* state of the function if a active function is ended *)
	xError : BOOL;					(* state of the function if a active function caused an error *)
	iErrorNr : INT;					(* state of the function if a active function caused an error, in this case give the error number *)
END_VAR
VAR
	xHardwareError: BOOL := FALSE;
	xInitError: BOOL := FALSE;
	iStepError: INT := 0;
	xStartMainCtr: BOOL := FALSE;
	xStartMainPrc: BOOL := FALSE;
	xInitMainCtr: BOOL := FALSE;
	iStepPrc: INT := 0;
	xSetEnd: BOOL := FALSE;
	xInitStep: BOOL := FALSE;
	xFreeze: BOOL := FALSE;
	iTmpErrorNr:INT:=0;
	xTmpInit:BOOL;
	iTmp:INT;
	xTmp: BOOL;
	TONWaitStop: TON;
END_VAR
(****************************************************************************************************************************************************)
(***********                                      This Functionblock define the function for start the toolrotation                                                    ************)
(****************************************************************************************************************************************************)

(******************************************************************************************************************************************)
(****************************				           Reset Function Part                                                 *****************************)
(******************************************************************************************************************************************)
IF xReset AND NOT(xSetEnd) THEN
	xEnd:=FALSE;
	xSetEnd:=TRUE;
END_IF;
(******************************************************************************************************************************************)
(****************************				              Error Controlling Part                                            *****************************)
(******************************************************************************************************************************************)
IF (xHardwareError OR ((TAxisToolLeft.T_CtrleSingle.xErr OR (TAxisToolCenter.T_CtrleSingle.xErr AND xMicroRodActive) OR TAxisToolRight.T_CtrleSingle.xErr OR (TAxisToolFeeder.T_CtrleSingle.xErr AND NOT(xMicroRodActive))) AND xStartMainPrc)) AND NOT(xSetEnd) THEN
	IF NOT(TAxisToolLeft.T_CtrleSingle.xExecute) AND ((NOT(TAxisToolCenter.T_CtrleSingle.xExecute) AND xMicroRodActive) OR NOT(xMicroRodActive)) AND NOT(TAxisToolRight.T_CtrleSingle.xExecute) AND ((NOT(TAxisToolFeeder.T_CtrleSingle.xExecute) AND NOT(xMicroRodActive)) OR xMicroRodActive) THEN
		IF NOT(xInitError) THEN
			iStepError:=100;
			xInitError:=TRUE;
			IF xHardwareError THEN
				iErrorNr:=iTmpErrorNr;
			ELSE
				xHardwareError:=TRUE;	(* Hardware Error *)
			END_IF;
		END_IF;
		CASE iStepError OF
			100:	iStepError:=0;
				xError:=TRUE;
		END_CASE;
		IF xQuitErr THEN
			xSetEnd:=TRUE;
		END_IF;
	END_IF;
END_IF;
(******************************************************************************************************************************************)
(****************************				              Main Controlling Part                                            *****************************)
(******************************************************************************************************************************************)
IF (xStart OR xStartMainCtr) AND NOT(xSetEnd) AND NOT(xHardwareError) THEN
	IF NOT (xInitMainCtr) THEN
		iTmpErrorNr:=0;
		iStepPrc:=100;
		xInitMainCtr:=TRUE;
		xStartMainCtr:=TRUE;
		xStart:=FALSE;
		xEnd:=FALSE;
		xAbord:=FALSE;
		xTmpInit:=FALSE;
	END_IF;
	IF xStop AND NOT(xTmpInit) THEN
		xTmpInit:=TRUE;
		iTmp:=100;
		RETURN;
	END_IF;
	IF xFreeze THEN
		IF xStart AND NOT(xAbord) THEN
			xFreeze:=FALSE;
			xStart:=FALSE;
		END_IF;
		IF xAbord THEN
			xAbord:=FALSE;
			xFreeze:=FALSE;
			xStart:=FALSE;
			xSetEnd:=TRUE;
		END_IF;
		RETURN;
	END_IF;
	IF NOT(xStartMainPrc) AND NOT(xSetEnd) THEN
		xStartMainPrc:=TRUE;
	END_IF;
END_IF;
(******************************************************************************************************************************************)
(****************************				             immediate Stop Part                                              *****************************)
(******************************************************************************************************************************************)
IF xTmpInit AND NOT(xSetEnd) THEN
	IF NOT(xSafetyCircuitOn) THEN
		xTmpInit:=FALSE;
		iTmp:=100;
		xSetEnd:=TRUE;
		RETURN;
	END_IF;
	CASE iTmp OF
		100:	IF TAxisToolLeft.T_CtrleSingle.xDone OR (TAxisToolCenter.T_CtrleSingle.xDone AND xMicroRodActive) OR TAxisToolRight.T_CtrleSingle.xDone OR (TAxisToolFeeder.T_CtrleSingle.xDone AND NOT(xMicroRodActive)) THEN
				TAxisToolLeft.T_CtrleSingle.iFunction:=5;
				TAxisToolLeft.T_CtrleSingle.xExecute:=TRUE;
				iTmp:=200;
			END_IF;
			RETURN;
		200:	IF NOT(TAxisToolLeft.T_CtrleSingle.xExecute) AND TAxisToolLeft.T_CtrleSingle.xDone THEN
				iTmp:=300;
				TONWaitStop(IN:=FALSE);
			END_IF;
			RETURN;
		300:	xTmp:=	((UINT_TO_WORD(TAxisToolRight.T_TxPdoParameter.uiStatusWord) AND 16#1000) = 16#1000) AND
					((((UINT_TO_WORD(TAxisToolCenter.T_TxPdoParameter.uiStatusWord) AND 16#1000) = 16#1000) AND xMicroRodActive) OR NOT(xMicroRodActive)) AND
					((((UINT_TO_WORD(TAxisToolFeeder.T_TxPdoParameter.uiStatusWord) AND 16#1000) = 16#1000) AND NOT(xMicroRodActive)) OR xMicroRodActive);
			TONWaitStop(IN:=TRUE,PT:=T#1000ms);
			IF TONWaitStop.Q AND xTmp THEN
				TONWaitStop(IN:=FALSE);
				iTmp:=400;
			END_IF;
			RETURN;
		400:	IF xMicroRodActive THEN
				IF TAxisToolCenter.T_CtrleSingle.xSlave THEN
					TAxisToolCenter.T_CtrleSingle.iFunction:=25;
					TAxisToolCenter.T_CtrleSingle.xExecute:=TRUE;
				END_IF;
			END_IF;
			IF TAxisToolRight.T_CtrleSingle.xSlave THEN
				TAxisToolRight.T_CtrleSingle.iFunction:=25;
				TAxisToolRight.T_CtrleSingle.xExecute:=TRUE;
			END_IF;
			IF NOT(xMicroRodActive) THEN
				IF TAxisToolFeeder.T_CtrleSingle.xSlave THEN
					TAxisToolFeeder.T_CtrleSingle.iFunction:=25;
					TAxisToolFeeder.T_CtrleSingle.xExecute:=TRUE;
				END_IF;
			END_IF;
			iTmp:=500;
			RETURN;
		500:	IF ((NOT(TAxisToolCenter.T_CtrleSingle.xExecute) AND TAxisToolCenter.T_CtrleSingle.xDone AND xMicroRodActive) OR NOT(xMicroRodActive)) AND
			    NOT(TAxisToolRight.T_CtrleSingle.xExecute) AND TAxisToolRight.T_CtrleSingle.xDone AND
			    ((NOT(TAxisToolFeeder.T_CtrleSingle.xExecute) AND TAxisToolFeeder.T_CtrleSingle.xDone AND NOT(xMicroRodActive)) OR xMicroRodActive) THEN
				xTmpInit:=FALSE;
				iTmp:=100;
				xSetEnd:=TRUE;
			END_IF;
			RETURN;
	END_CASE;
END_IF;
(******************************************************************************************************************************************)
(****************************				             Main Procedure Part                                             *****************************)
(******************************************************************************************************************************************)
IF xStartMainPrc AND NOT(xSetEnd) AND NOT(xHardwareError) THEN
	CASE iStepPrc OF
		100:	IF NOT(xInitStep) THEN
				xInitStep:=TRUE;
				IF NOT(TAxisToolLeft.T_CtrleSingle.xDone) OR (NOT(TAxisToolCenter.T_CtrleSingle.xDone) AND xMicroRodActive) OR NOT(TAxisToolRight.T_CtrleSingle.xDone) OR (NOT(TAxisToolFeeder.T_CtrleSingle.xDone) AND NOT(xMicroRodActive)) THEN
					xHardwareError:=TRUE;
					iTmpErrorNr:=1;
					RETURN;
				END_IF;
				IF NOT(TAxisToolLeft.T_CtrleSingle.xPower) THEN
					TAxisToolLeft.T_CtrleSingle.iFunction:=3;
					TAxisToolLeft.T_CtrleSingle.xExecute:=TRUE;
				END_IF;
				IF xMicroRodActive THEN
					IF NOT(TAxisToolCenter.T_CtrleSingle.xPower) THEN
						TAxisToolCenter.T_CtrleSingle.iFunction:=3;
						TAxisToolCenter.T_CtrleSingle.xExecute:=TRUE;
					END_IF;
				END_IF;
				IF NOT(TAxisToolRight.T_CtrleSingle.xPower) THEN
					TAxisToolRight.T_CtrleSingle.iFunction:=3;
					TAxisToolRight.T_CtrleSingle.xExecute:=TRUE;
				END_IF;
				IF NOT(xMicroRodActive) THEN
					IF NOT(TAxisToolFeeder.T_CtrleSingle.xPower) THEN
						TAxisToolFeeder.T_CtrleSingle.iFunction:=3;
						TAxisToolFeeder.T_CtrleSingle.xExecute:=TRUE;
					END_IF;
				END_IF;
			END_IF;
			IF NOT(TAxisToolLeft.T_CtrleSingle.xExecute) AND TAxisToolLeft.T_CtrleSingle.xDone AND
			    ((NOT(TAxisToolCenter.T_CtrleSingle.xExecute) AND TAxisToolCenter.T_CtrleSingle.xDone AND xMicroRodActive) OR NOT(xMicroRodActive)) AND
			    NOT(TAxisToolRight.T_CtrleSingle.xExecute) AND TAxisToolRight.T_CtrleSingle.xDone AND
			    ((NOT(TAxisToolFeeder.T_CtrleSingle.xExecute) AND TAxisToolFeeder.T_CtrleSingle.xDone AND NOT(xMicroRodActive)) OR xMicroRodActive) THEN
				xStartMainPrc:=FALSE;
				xInitStep:=FALSE;
				iStepPrc:=200;
			END_IF;
		200:	IF NOT(xInitStep) THEN
				xInitStep:=TRUE;
				IF xMicroRodActive THEN
					IF NOT(TAxisToolCenter.T_CtrleSingle.xSlave) THEN
						TAxisToolCenter.T_CtrleSingle.iFunction:=25;
						TAxisToolCenter.T_CtrleSingle.xExecute:=TRUE;
					END_IF;
				END_IF;
				IF NOT(TAxisToolRight.T_CtrleSingle.xSlave) THEN
					TAxisToolRight.T_CtrleSingle.iFunction:=25;
					TAxisToolRight.T_CtrleSingle.xExecute:=TRUE;
				END_IF;
				IF NOT(xMicroRodActive) THEN
					IF NOT(TAxisToolFeeder.T_CtrleSingle.xSlave) THEN
						TAxisToolFeeder.T_CtrleSingle.iFunction:=25;
						TAxisToolFeeder.T_CtrleSingle.xExecute:=TRUE;
					END_IF;
				END_IF;
			END_IF;
			IF ((NOT(TAxisToolCenter.T_CtrleSingle.xExecute) AND TAxisToolCenter.T_CtrleSingle.xDone AND xMicroRodActive) OR NOT(xMicroRodActive)) AND
			    NOT(TAxisToolRight.T_CtrleSingle.xExecute) AND TAxisToolRight.T_CtrleSingle.xDone AND
			    ((NOT(TAxisToolFeeder.T_CtrleSingle.xExecute) AND TAxisToolFeeder.T_CtrleSingle.xDone AND NOT(xMicroRodActive)) OR xMicroRodActive) THEN
				xStartMainPrc:=FALSE;
				xInitStep:=FALSE;
				iStepPrc:=300;
			END_IF;
		300:	IF NOT(xInitStep) THEN
				xInitStep:=TRUE;
				TAxisToolLeft.T_CtrleSingle.iFunction:=6;
				TAxisToolLeft.T_CtrleSingle.xExecute:=TRUE;
			END_IF;
			IF NOT(TAxisToolLeft.T_CtrleSingle.xExecute) AND TAxisToolLeft.T_CtrleSingle.xDone THEN
				xStartMainPrc:=FALSE;
				xInitStep:=FALSE;
				iStepPrc:=0;
				xSetEnd:=TRUE;
			END_IF;
	END_CASE;
END_IF;
(******************************************************************************************************************************************)
(****************************				           Parallel Procedure Part                                          *****************************)
(******************************************************************************************************************************************)

(******************************************************************************************************************************************)
(****************************				             	Init / Reset Part                                                   *****************************)
(******************************************************************************************************************************************)
IF xSetEnd THEN
	xEnd:=TRUE;
	xInitStep:=FALSE;
	xSetEnd:=FALSE;
	xStop:=FALSE;
	xStartMainPrc:=FALSE;
	xInitMainCtr:=FALSE;
	xStartMainCtr:=FALSE;
	xStart:=FALSE;
	xHardwareError:=FALSE;
	xQuitErr:=FALSE;
	xError:=FALSE;
	iErrorNr:=0;
	xInitError:=FALSE;
	xFreeze:=FALSE;
	xAbord:=FALSE;
	xReset:=FALSE;
END_IF;
END_FUNCTION_BLOCK

(* POU PRG_STATION_LAYER3/FB_STATIONEN/FB_FUNCTION/FB_FctToolRotationTorqueStop, ST *)
FUNCTION_BLOCK FB_FctToolRotationTorqueStop
VAR_INPUT
	xMicroRodActive: BOOL;		(* choice of the machine MicroWire or MicroRod *)
	xBeckhoffDriveActive: BOOL;	(* choice of the axis Beckhoff or EcoStep *)
	xSafetyCircuitOn:BOOL;			(* state of the safety circuit-->TRUE=Machine current ON, FALSE=Machine current OFF *)
END_VAR
VAR_IN_OUT
	xStart : BOOL;					(* start the function *)
	xReset : BOOL;				(* reset the function *)
	xStop : BOOL;					(* stop the active function *)
	xQuitErr : BOOL;				(* quit the error caused of the active function *)
	xAbord : BOOL;				(* abord the active function *)
	TAxisToolLeft:ST_AXIS;		(* data structure for the ToolLeft axis *)
	TAxisToolCenter:ST_AXIS;		(* data structure for the ToolCenter axis *)
	TAxisToolRight:ST_AXIS;		(* data structure for the ToolRight axis *)
	TAxisToolFeeder:ST_AXIS;		(* data structure for the ToolFeeder axis *)
END_VAR
VAR_OUTPUT
	xEnd : BOOL;					(* state of the function if a active function is ended *)
	xError : BOOL;					(* state of the function if a active function caused an error *)
	iErrorNr : INT;					(* state of the function if a active function caused an error, in this case give the error number *)
END_VAR
VAR
	xHardwareError: BOOL := FALSE;
	xInitError: BOOL := FALSE;
	iStepError: INT := 0;
	xStartMainCtr: BOOL := FALSE;
	xStartMainPrc: BOOL := FALSE;
	xInitMainCtr: BOOL := FALSE;
	iStepPrc: INT := 0;
	xSetEnd: BOOL := FALSE;
	xInitStep: BOOL := FALSE;
	xFreeze: BOOL := FALSE;
	iTmpErrorNr:INT:=0;
	xTmpInit:BOOL;
	iTmp:INT;
	xTmp: BOOL;
	TONWaitStop: TON;
END_VAR
(****************************************************************************************************************************************************)
(***********                                      This Functionblock define the function for stop the toolrotation                                                    ************)
(****************************************************************************************************************************************************)

(******************************************************************************************************************************************)
(****************************				           Reset Function Part                                                 *****************************)
(******************************************************************************************************************************************)
IF xReset AND NOT(xSetEnd) THEN
	xEnd:=FALSE;
	xSetEnd:=TRUE;
END_IF;
(******************************************************************************************************************************************)
(****************************				              Error Controlling Part                                            *****************************)
(******************************************************************************************************************************************)
IF (xHardwareError OR ((TAxisToolLeft.T_CtrleSingle.xErr OR (TAxisToolCenter.T_CtrleSingle.xErr AND xMicroRodActive) OR TAxisToolRight.T_CtrleSingle.xErr OR (TAxisToolFeeder.T_CtrleSingle.xErr AND NOT(xMicroRodActive))) AND xStartMainPrc)) AND NOT(xSetEnd) THEN
	IF NOT(TAxisToolLeft.T_CtrleSingle.xExecute) AND ((NOT(TAxisToolCenter.T_CtrleSingle.xExecute) AND xMicroRodActive) OR NOT(xMicroRodActive)) AND NOT(TAxisToolRight.T_CtrleSingle.xExecute) AND ((NOT(TAxisToolFeeder.T_CtrleSingle.xExecute) AND NOT(xMicroRodActive)) OR xMicroRodActive) THEN
		IF NOT(xInitError) THEN
			iStepError:=100;
			xInitError:=TRUE;
			IF xHardwareError THEN
				iErrorNr:=iTmpErrorNr;
			ELSE
				xHardwareError:=TRUE;	(* Hardware Error *)
			END_IF;
		END_IF;
		CASE iStepError OF
			100:	iStepError:=0;
				xError:=TRUE;
		END_CASE;
		IF xQuitErr THEN
			xSetEnd:=TRUE;
		END_IF;
	END_IF;
END_IF;
(******************************************************************************************************************************************)
(****************************				              Main Controlling Part                                            *****************************)
(******************************************************************************************************************************************)
IF (xStart OR xStartMainCtr) AND NOT(xSetEnd) AND NOT(xHardwareError) THEN
	IF NOT (xInitMainCtr) THEN
		iTmpErrorNr:=0;
		iStepPrc:=100;
		xInitMainCtr:=TRUE;
		xStartMainCtr:=TRUE;
		xStart:=FALSE;
		xEnd:=FALSE;
		xAbord:=FALSE;
		xTmpInit:=FALSE;
	END_IF;
	IF xStop AND NOT(xTmpInit) THEN
		xTmpInit:=TRUE;
		iTmp:=100;
		RETURN;
	END_IF;
	IF xFreeze THEN
		IF xStart AND NOT(xAbord) THEN
			xFreeze:=FALSE;
			xStart:=FALSE;
		END_IF;
		IF xAbord THEN
			xAbord:=FALSE;
			xFreeze:=FALSE;
			xStart:=FALSE;
			xSetEnd:=TRUE;
		END_IF;
		RETURN;
	END_IF;
	IF NOT(xStartMainPrc) AND NOT(xSetEnd) THEN
		xStartMainPrc:=TRUE;
	END_IF;
END_IF;
(******************************************************************************************************************************************)
(****************************				             immediate Stop Part                                              *****************************)
(******************************************************************************************************************************************)
IF xTmpInit AND NOT(xSetEnd) THEN
	IF NOT(xSafetyCircuitOn) THEN
		xTmpInit:=FALSE;
		iTmp:=100;
		xSetEnd:=TRUE;
		RETURN;
	END_IF;
	CASE iTmp OF
		(* No immediately stopping *)
		100:	xTmpInit:=FALSE;
			iTmp:=100;
	END_CASE;
END_IF;
(******************************************************************************************************************************************)
(****************************				             Main Procedure Part                                             *****************************)
(******************************************************************************************************************************************)
IF xStartMainPrc AND NOT(xSetEnd) AND NOT(xHardwareError) THEN
	CASE iStepPrc OF
		100:	IF NOT(xInitStep) THEN
				xInitStep:=TRUE;
				IF NOT(TAxisToolLeft.T_CtrleSingle.xDone) OR (NOT(TAxisToolCenter.T_CtrleSingle.xDone) AND xMicroRodActive) OR NOT(TAxisToolRight.T_CtrleSingle.xDone) OR (NOT(TAxisToolFeeder.T_CtrleSingle.xDone) AND NOT(xMicroRodActive)) THEN
					xHardwareError:=TRUE;
					iTmpErrorNr:=1;
					RETURN;
				END_IF;
				TAxisToolLeft.T_CtrleSingle.iFunction:=5;
				TAxisToolLeft.T_CtrleSingle.xExecute:=TRUE;
			END_IF;
			IF NOT(TAxisToolLeft.T_CtrleSingle.xExecute) AND TAxisToolLeft.T_CtrleSingle.xDone THEN
				xStartMainPrc:=FALSE;
				xInitStep:=FALSE;
				iStepPrc:=199;
			END_IF;
		199:	xTmp:=	((UINT_TO_WORD(TAxisToolRight.T_TxPdoParameter.uiStatusWord) AND 16#1000) = 16#1000) AND
					((((UINT_TO_WORD(TAxisToolCenter.T_TxPdoParameter.uiStatusWord) AND 16#1000) = 16#1000) AND xMicroRodActive) OR NOT(xMicroRodActive)) AND
					((((UINT_TO_WORD(TAxisToolFeeder.T_TxPdoParameter.uiStatusWord) AND 16#1000) = 16#1000) AND NOT(xMicroRodActive)) OR xMicroRodActive);
			IF NOT(xInitStep) THEN
				xInitStep:=TRUE;
				TONWaitStop(IN:=FALSE);
			END_IF;
			TONWaitStop(IN:=TRUE,PT:=T#1000ms);
			IF TONWaitStop.Q AND xTmp THEN
				TONWaitStop(IN:=FALSE);
				xStartMainPrc:=FALSE;
				xInitStep:=FALSE;
				iStepPrc:=200;
			END_IF;
		200:	IF NOT(xInitStep) THEN
				xInitStep:=TRUE;
				IF xMicroRodActive THEN
					IF TAxisToolCenter.T_CtrleSingle.xSlave THEN
						TAxisToolCenter.T_CtrleSingle.iFunction:=25;
						TAxisToolCenter.T_CtrleSingle.xExecute:=TRUE;
					END_IF;
				END_IF;
				IF TAxisToolRight.T_CtrleSingle.xSlave THEN
					TAxisToolRight.T_CtrleSingle.iFunction:=25;
					TAxisToolRight.T_CtrleSingle.xExecute:=TRUE;
				END_IF;
				IF NOT(xMicroRodActive) THEN
					IF TAxisToolFeeder.T_CtrleSingle.xSlave THEN
						TAxisToolFeeder.T_CtrleSingle.iFunction:=25;
						TAxisToolFeeder.T_CtrleSingle.xExecute:=TRUE;
					END_IF;
				END_IF;
			END_IF;
			IF ((NOT(TAxisToolCenter.T_CtrleSingle.xExecute) AND TAxisToolCenter.T_CtrleSingle.xDone AND xMicroRodActive) OR NOT(xMicroRodActive)) AND
			    NOT(TAxisToolRight.T_CtrleSingle.xExecute) AND TAxisToolRight.T_CtrleSingle.xDone AND
			    ((NOT(TAxisToolFeeder.T_CtrleSingle.xExecute) AND TAxisToolFeeder.T_CtrleSingle.xDone AND NOT(xMicroRodActive)) OR xMicroRodActive) THEN
				xStartMainPrc:=FALSE;
				xInitStep:=FALSE;
				iStepPrc:=0;
				xSetEnd:=TRUE;
			END_IF;
	END_CASE;
END_IF;
(******************************************************************************************************************************************)
(****************************				           Parallel Procedure Part                                          *****************************)
(******************************************************************************************************************************************)

(******************************************************************************************************************************************)
(****************************				             	Init / Reset Part                                                   *****************************)
(******************************************************************************************************************************************)
IF xSetEnd THEN
	xEnd:=TRUE;
	xInitStep:=FALSE;
	xSetEnd:=FALSE;
	xStop:=FALSE;
	xStartMainPrc:=FALSE;
	xInitMainCtr:=FALSE;
	xStartMainCtr:=FALSE;
	xStart:=FALSE;
	xHardwareError:=FALSE;
	xQuitErr:=FALSE;
	xError:=FALSE;
	iErrorNr:=0;
	xInitError:=FALSE;
	xFreeze:=FALSE;
	xAbord:=FALSE;
	xReset:=FALSE;
END_IF;
END_FUNCTION_BLOCK

(* POU PRG_STATION_LAYER3/FB_STATIONEN/FB_FUNCTION/FB_FctGrindFeedAbsRelPosition, ST *)
FUNCTION_BLOCK FB_FctGrindFeedAbsRelPosition
VAR_INPUT
	xMicroRodActive: BOOL;		(* choice of the machine MicroWire or MicroRod *)
	xBeckhoffDriveActive: BOOL;	(* choice of the axis Beckhoff or EcoStep *)
	xSafetyCircuitOn:BOOL;			(* state of the safety circuit-->TRUE=Machine current ON, FALSE=Machine current OFF *)
	iFunctionNr:INT;				(* state of the called function number-->4=move axis absolut, 5=move axis relative *)
END_VAR
VAR_IN_OUT
	xStart : BOOL;					(* start the function *)
	xReset : BOOL;				(* reset the function *)
	xStop : BOOL;					(* stop the active function *)
	xQuitErr : BOOL;				(* quit the error caused of the active function *)
	xAbord : BOOL;				(* abord the active function *)
	TAxisGrindFeeder:ST_AXIS;	(* data structure for the GrindFeeder axis *)
END_VAR
VAR_OUTPUT
	xEnd : BOOL;					(* state of the function if a active function is ended *)
	xError : BOOL;					(* state of the function if a active function caused an error *)
	iErrorNr : INT;					(* state of the function if a active function caused an error, in this case give the error number *)
END_VAR
VAR
	xHardwareError: BOOL := FALSE;
	xInitError: BOOL := FALSE;
	iStepError: INT := 0;
	xStartMainCtr: BOOL := FALSE;
	xStartMainPrc: BOOL := FALSE;
	xInitMainCtr: BOOL := FALSE;
	iStepPrc: INT := 0;
	xSetEnd: BOOL := FALSE;
	xInitStep: BOOL := FALSE;
	xFreeze: BOOL := FALSE;
	iTmpErrorNr:INT:=0;
	xTmpInit:BOOL;
	iTmp:INT;
END_VAR
(****************************************************************************************************************************************************)
(***********       This Functionblock define the function for set the GrindFeeder Axis to the relative or absolut position       ************)
(****************************************************************************************************************************************************)

(******************************************************************************************************************************************)
(****************************				           Reset Function Part                                                 *****************************)
(******************************************************************************************************************************************)
IF xReset AND NOT(xSetEnd) THEN
	xEnd:=FALSE;
	xSetEnd:=TRUE;
END_IF;
(******************************************************************************************************************************************)
(****************************				              Error Controlling Part                                            *****************************)
(******************************************************************************************************************************************)
IF (xHardwareError OR ((TAxisGrindFeeder.T_CtrleSingle.xErr) AND xStartMainPrc)) AND NOT(xSetEnd) THEN
	IF NOT(TAxisGrindFeeder.T_CtrleSingle.xExecute) THEN
		IF NOT(xInitError) THEN
			iStepError:=100;
			xInitError:=TRUE;
			IF xHardwareError THEN
				iErrorNr:=iTmpErrorNr;
			ELSE
				xHardwareError:=TRUE;	(* Hardware Error *)
			END_IF;
		END_IF;
		CASE iStepError OF
			100:	iStepError:=0;
				xError:=TRUE;
		END_CASE;
		IF xQuitErr THEN
			xSetEnd:=TRUE;
		END_IF;
	END_IF;
END_IF;
(******************************************************************************************************************************************)
(****************************				              Main Controlling Part                                            *****************************)
(******************************************************************************************************************************************)
IF (xStart OR xStartMainCtr) AND NOT(xSetEnd) AND NOT(xHardwareError) THEN
	IF NOT (xInitMainCtr) THEN
		iTmpErrorNr:=0;
		iStepPrc:=100;
		xInitMainCtr:=TRUE;
		xStartMainCtr:=TRUE;
		xStart:=FALSE;
		xEnd:=FALSE;
		xAbord:=FALSE;
		xTmpInit:=FALSE;
	END_IF;
	IF xStop AND NOT(xTmpInit) THEN
		xTmpInit:=TRUE;
		iTmp:=100;
		RETURN;
	END_IF;
	IF xFreeze THEN
		IF xStart AND NOT(xAbord) THEN
			xFreeze:=FALSE;
			xStart:=FALSE;
		END_IF;
		IF xAbord THEN
			xAbord:=FALSE;
			xFreeze:=FALSE;
			xStart:=FALSE;
			xSetEnd:=TRUE;
		END_IF;
		RETURN;
	END_IF;
	IF NOT(xStartMainPrc) AND NOT(xSetEnd) THEN
		xStartMainPrc:=TRUE;
	END_IF;
END_IF;
(******************************************************************************************************************************************)
(****************************				             immediate Stop Part                                              *****************************)
(******************************************************************************************************************************************)
IF xTmpInit AND NOT(xSetEnd) THEN
	IF NOT(xSafetyCircuitOn) THEN
		xTmpInit:=FALSE;
		iTmp:=100;
		xSetEnd:=TRUE;
		RETURN;
	END_IF;
	CASE iTmp OF
		100:	TAxisGrindFeeder.T_CtrleSingle.iFunction:=5;
			TAxisGrindFeeder.T_CtrleSingle.xExecute:=TRUE;
			iTmp:=200;
			RETURN;
		200:	IF NOT(TAxisGrindFeeder.T_CtrleSingle.xExecute) AND TAxisGrindFeeder.T_CtrleSingle.xDone THEN
				iTmp:=300;
			END_IF;
			RETURN;
		300:	xTmpInit:=FALSE;
			iTmp:=100;
			xSetEnd:=TRUE;
			RETURN;
	END_CASE;
END_IF;
(******************************************************************************************************************************************)
(****************************				             Main Procedure Part                                             *****************************)
(******************************************************************************************************************************************)
IF xStartMainPrc AND NOT(xSetEnd) AND NOT(xHardwareError) THEN
	CASE iStepPrc OF
		100:	IF NOT(xInitStep) THEN
				xInitStep:=TRUE;
				IF NOT(TAxisGrindFeeder.T_CtrleSingle.xDone)THEN
					xHardwareError:=TRUE;
					iTmpErrorNr:=1;
					RETURN;
				END_IF;
				IF NOT(TAxisGrindFeeder.T_CtrleSingle.xPower) THEN
					TAxisGrindFeeder.T_CtrleSingle.iFunction:=3;
					TAxisGrindFeeder.T_CtrleSingle.xExecute:=TRUE;
				END_IF;
			END_IF;
			IF NOT(TAxisGrindFeeder.T_CtrleSingle.xExecute) AND TAxisGrindFeeder.T_CtrleSingle.xDone THEN
				xStartMainPrc:=FALSE;
				xInitStep:=FALSE;
				iStepPrc:=200;
			END_IF;
		200:	IF NOT(xInitStep) THEN
				xInitStep:=TRUE;
				IF (iFunctionNr = 4) THEN
					TAxisGrindFeeder.T_CtrleSingle.iFunction:=7;	(* Move Absolut *)
				END_IF;
				IF (iFunctionNr = 5) THEN
					TAxisGrindFeeder.T_CtrleSingle.iFunction:=8;	(* Move Relative *)
				END_IF;
				TAxisGrindFeeder.T_CtrleSingle.xExecute:=TRUE;
			END_IF;
			IF NOT(TAxisGrindFeeder.T_CtrleSingle.xExecute) AND TAxisGrindFeeder.T_CtrleSingle.xDone THEN
				xStartMainPrc:=FALSE;
				xInitStep:=FALSE;
				iStepPrc:=0;
				xSetEnd:=TRUE;
			END_IF;
	END_CASE;
END_IF;
(******************************************************************************************************************************************)
(****************************				           Parallel Procedure Part                                          *****************************)
(******************************************************************************************************************************************)

(******************************************************************************************************************************************)
(****************************				             	Init / Reset Part                                                   *****************************)
(******************************************************************************************************************************************)
IF xSetEnd THEN
	xEnd:=TRUE;
	xInitStep:=FALSE;
	xSetEnd:=FALSE;
	xStop:=FALSE;
	xStartMainPrc:=FALSE;
	xInitMainCtr:=FALSE;
	xStartMainCtr:=FALSE;
	xStart:=FALSE;
	xHardwareError:=FALSE;
	xQuitErr:=FALSE;
	xError:=FALSE;
	iErrorNr:=0;
	xInitError:=FALSE;
	xFreeze:=FALSE;
	xAbord:=FALSE;
	xReset:=FALSE;
END_IF;
END_FUNCTION_BLOCK

(* POU PRG_STATION_LAYER3/FB_STATIONEN/FB_FUNCTION/FB_FctSetAxisPosition, ST *)
FUNCTION_BLOCK FB_FctSetAxisPosition
VAR_INPUT
	xMicroRodActive: BOOL;		(* choice of the machine MicroWire or MicroRod *)
	xBeckhoffDriveActive: BOOL;	(* choice of the axis Beckhoff or EcoStep *)
	xSafetyCircuitOn:BOOL;			(* state of the safety circuit-->TRUE=Machine current ON, FALSE=Machine current OFF *)
	iFunctionNr:INT;				(* state of the called function number-->	6=set position of the ToolLeft axis
																	7=set position of the ToolCenter axis
																	8=set position of the ToolRight axis
																	9=set position of the ToolFeeder axis
																	10=set position of the GrindFeeder axis *)
END_VAR
VAR_IN_OUT
	xStart : BOOL;					(* start the function *)
	xReset : BOOL;				(* reset the function *)
	xStop : BOOL;					(* stop the active function *)
	xQuitErr : BOOL;				(* quit the error caused of the active function *)
	xAbord : BOOL;				(* abord the active function *)
	TAxisToolLeft:ST_AXIS;		(* data structure for the ToolLeft axis *)
	TAxisToolCenter:ST_AXIS;		(* data structure for the ToolCenter axis *)
	TAxisToolRight:ST_AXIS;		(* data structure for the ToolRight axis *)
	TAxisToolFeeder:ST_AXIS;		(* data structure for the ToolFeeder axis *)
	TAxisGrindFeeder:ST_AXIS;	(* data structure for the GrindFeeder axis *)
END_VAR
VAR_OUTPUT
	xEnd : BOOL;					(* state of the function if a active function is ended *)
	xError : BOOL;					(* state of the function if a active function caused an error *)
	iErrorNr : INT;					(* state of the function if a active function caused an error, in this case give the error number *)
END_VAR
VAR
	xHardwareError: BOOL := FALSE;
	xInitError: BOOL := FALSE;
	iStepError: INT := 0;
	xStartMainCtr: BOOL := FALSE;
	xStartMainPrc: BOOL := FALSE;
	xInitMainCtr: BOOL := FALSE;
	iStepPrc: INT := 0;
	xSetEnd: BOOL := FALSE;
	xInitStep: BOOL := FALSE;
	xFreeze: BOOL := FALSE;
	iTmpErrorNr:INT:=0;
	xTmpInit:BOOL;
	iTmp:INT;
	ptrTAxis: POINTER TO ST_AXIS;
	xReadFirstTime: BOOL;
END_VAR
(****************************************************************************************************************************************************)
(***********       This Functionblock set a position for the ToolLeft,ToolCenter,ToolRight,ToolFeeder or GrindFeeder       ************)
(****************************************************************************************************************************************************)

IF NOT(xReadFirstTime) THEN
	xReadFirstTime:=TRUE;
	ptrTAxis:=ADR(TAxisToolLeft);
END_IF;
(******************************************************************************************************************************************)
(****************************				           Reset Function Part                                                 *****************************)
(******************************************************************************************************************************************)
IF xReset AND NOT(xSetEnd) THEN
	ptrTAxis:=ADR(TAxisToolLeft);
	xEnd:=FALSE;
	xSetEnd:=TRUE;
END_IF;
(******************************************************************************************************************************************)
(****************************				              Error Controlling Part                                            *****************************)
(******************************************************************************************************************************************)
IF (xHardwareError OR ((ptrTAxis^.T_CtrleSingle.xErr) AND xStartMainPrc)) AND NOT(xSetEnd) THEN
	IF NOT(ptrTAxis^.T_CtrleSingle.xExecute) THEN
		IF NOT(xInitError) THEN
			iStepError:=100;
			xInitError:=TRUE;
			IF xHardwareError THEN
				iErrorNr:=iTmpErrorNr;
			ELSE
				xHardwareError:=TRUE;	(* Hardware Error *)
			END_IF;
		END_IF;
		CASE iStepError OF
			100:	iStepError:=0;
				xError:=TRUE;
		END_CASE;
		IF xQuitErr THEN
			xSetEnd:=TRUE;
		END_IF;
	END_IF;
END_IF;
(******************************************************************************************************************************************)
(****************************				              Main Controlling Part                                            *****************************)
(******************************************************************************************************************************************)
IF (xStart OR xStartMainCtr) AND NOT(xSetEnd) AND NOT(xHardwareError) THEN
	IF NOT (xInitMainCtr) THEN
		IF (iFunctionNr = 6) THEN
			ptrTAxis:=ADR(TAxisToolLeft);
		ELSIF (iFunctionNr = 7) THEN
			ptrTAxis:=ADR(TAxisToolCenter);
		ELSIF (iFunctionNr = 8) THEN
			ptrTAxis:=ADR(TAxisToolRight);
		ELSIF (iFunctionNr = 9) THEN
			ptrTAxis:=ADR(TAxisToolFeeder);
		ELSIF (iFunctionNr = 10) THEN
			ptrTAxis:=ADR(TAxisGrindFeeder);
		ELSE
			ptrTAxis:=ADR(TAxisToolLeft);
		END_IF;
		iTmpErrorNr:=0;
		iStepPrc:=100;
		xInitMainCtr:=TRUE;
		xStartMainCtr:=TRUE;
		xStart:=FALSE;
		xEnd:=FALSE;
		xAbord:=FALSE;
		xTmpInit:=FALSE;
	END_IF;
	IF xStop AND NOT(xTmpInit) THEN
		xTmpInit:=TRUE;
		iTmp:=100;
		RETURN;
	END_IF;
	IF xFreeze THEN
		IF xStart AND NOT(xAbord) THEN
			xFreeze:=FALSE;
			xStart:=FALSE;
		END_IF;
		IF xAbord THEN
			xAbord:=FALSE;
			xFreeze:=FALSE;
			xStart:=FALSE;
			xSetEnd:=TRUE;
		END_IF;
		RETURN;
	END_IF;
	IF NOT(xStartMainPrc) AND NOT(xSetEnd) THEN
		xStartMainPrc:=TRUE;
	END_IF;
END_IF;
(******************************************************************************************************************************************)
(****************************				             immediate Stop Part                                              *****************************)
(******************************************************************************************************************************************)
IF xTmpInit AND NOT(xSetEnd) THEN
	IF NOT(xSafetyCircuitOn) THEN
		xTmpInit:=FALSE;
		iTmp:=100;
		xSetEnd:=TRUE;
		RETURN;
	END_IF;
	CASE iTmp OF
		100:	IF NOT(ptrTAxis^.T_CtrleSingle.xDone) THEN
				ptrTAxis^.T_CtrleSingle.xReset:=TRUE;
				iTmp:=200;
			END_IF;
			RETURN;
		200:	IF NOT(ptrTAxis^.T_CtrleSingle.xReset) AND ptrTAxis^.T_CtrleSingle.xDone THEN
				iTmp:=300;
			END_IF;
			RETURN;
		300:	xTmpInit:=FALSE;
			iTmp:=100;
			xSetEnd:=TRUE;
			RETURN;
	END_CASE;
END_IF;
(******************************************************************************************************************************************)
(****************************				             Main Procedure Part                                             *****************************)
(******************************************************************************************************************************************)
IF xStartMainPrc AND NOT(xSetEnd) AND NOT(xHardwareError) THEN
	CASE iStepPrc OF
		100:	IF NOT(xInitStep) THEN
				xInitStep:=TRUE;
				IF NOT(ptrTAxis^.T_CtrleSingle.xDone)THEN
					xHardwareError:=TRUE;
					iTmpErrorNr:=1;
					RETURN;
				END_IF;
				ptrTAxis^.T_CtrleSingle.iFunction:=11;
				ptrTAxis^.T_CtrleSingle.xExecute:=TRUE;
			END_IF;
			IF NOT(ptrTAxis^.T_CtrleSingle.xExecute) AND ptrTAxis^.T_CtrleSingle.xDone THEN
				xStartMainPrc:=FALSE;
				xInitStep:=FALSE;
				iStepPrc:=0;
				xSetEnd:=TRUE;
			END_IF;
	END_CASE;
END_IF;
(******************************************************************************************************************************************)
(****************************				           Parallel Procedure Part                                          *****************************)
(******************************************************************************************************************************************)

(******************************************************************************************************************************************)
(****************************				             	Init / Reset Part                                                   *****************************)
(******************************************************************************************************************************************)
IF xSetEnd THEN
	xEnd:=TRUE;
	xInitStep:=FALSE;
	xSetEnd:=FALSE;
	xStop:=FALSE;
	xStartMainPrc:=FALSE;
	xInitMainCtr:=FALSE;
	xStartMainCtr:=FALSE;
	xStart:=FALSE;
	xHardwareError:=FALSE;
	xQuitErr:=FALSE;
	xError:=FALSE;
	iErrorNr:=0;
	xInitError:=FALSE;
	xFreeze:=FALSE;
	xAbord:=FALSE;
	xReset:=FALSE;
END_IF;
END_FUNCTION_BLOCK

(* POU PRG_STATION_LAYER3/FB_STATIONEN/FB_FUNCTION/FB_FctToolWorkingGeometry, ST *)
FUNCTION_BLOCK FB_FctToolWorkingGeometry
VAR_INPUT
	xMicroRodActive: BOOL;		(* choice of the machine MicroWire or MicroRod *)
	xBeckhoffDriveActive: BOOL;	(* choice of the axis Beckhoff or EcoStep *)
	xSafetyCircuitOn:BOOL;			(* state of the safety circuit-->TRUE=Machine current ON, FALSE=Machine current OFF *)
	T_ProcessImageData:ST_RETAIN_DATA_PROCESSIMAGE;	(* Novram data structure for the process parameter *)
	T_Standard:ST_RETAIN_DATA;							(* Novram data structure for the standard process parameter *)
END_VAR
VAR_IN_OUT
	xStart : BOOL;					(* start the function *)
	xReset : BOOL;				(* reset the function *)
	xStop : BOOL;					(* stop the active function *)
	xQuitErr : BOOL;				(* quit the error caused of the active function *)
	xAbord : BOOL;				(* abord the active function *)
	TAxisToolLeft:ST_AXIS;		(* data structure for the ToolLeft axis *)
	TAxisToolCenter:ST_AXIS;		(* data structure for the ToolCenter axis *)
	TAxisToolRight:ST_AXIS;		(* data structure for the ToolRight axis *)
	TAxisToolFeeder:ST_AXIS;		(* data structure for the ToolFeeder axis *)
	TAxisGrindFeeder:ST_AXIS;	(* data structure for the GrindFeeder axis *)
	T_WorkTool:ST_WORKTOOL;	(* Tool parameter *)
END_VAR
VAR_OUTPUT
	xEnd : BOOL;					(* state of the function if a active function is ended *)
	xError : BOOL;					(* state of the function if a active function caused an error *)
	iErrorNr : INT;					(* state of the function if a active function caused an error, in this case give the error number *)
	bActivePartNumber:BYTE;		(* gives the active number of the worked section of the geometry *)
	lrProcessToolFeederActualPosition:LREAL;	(* gives the calculated position of the ToolFeeder *)
	lrProcessToolFeederSpeed:LREAL;			(* gives the calculated speed of the ToolFeeder *)
	iCountDownPlungeCycle:INT;
END_VAR
VAR
	xHardwareError: BOOL := FALSE;
	xInitError: BOOL := FALSE;
	iStepError: INT := 0;
	xStartMainCtr: BOOL := FALSE;
	xStartMainPrc: BOOL := FALSE;
	xInitMainCtr: BOOL := FALSE;
	iStepPrc: INT := 0;
	xSetEnd: BOOL := FALSE;
	xInitStep: BOOL := FALSE;
	xFreeze: BOOL := FALSE;
	iTmpErrorNr:INT:=0;
	xTmpInit:BOOL;
	iTmp:INT;
	xTmp: BOOL;
	xReadFirstTime: BOOL;
	xTmp1: BOOL;
	rToolRotationSpeed: REAL;
	FBToolCalcul:FB_TOOL_CALCUL_NEW;

	rToolFeedLength: REAL;
	rToolDiameter: REAL;
	rGrindFeedPlunge: REAL;
	ii: INT;
	iStartSection: INT;
	iEndSection: INT;
	rSpeedGrindFeed: REAL;
	rSpeedToolFeed: REAL;
	rTimeGrindPlunge: REAL;
	FBCalcGearFactor: FB_CALC_GEARFACTOR;
	lrToolFeederActualPosition: LREAL;
	iTmpStartSection: INT;
	FBCalcPlungeGrinding: FB_CALC_PLUNGE_GRINDING;
	xResetFB: BOOL;
	xGrindFeedMaster: BOOL;
	xCheckToolFeedPosition: BOOL;
	lrToolFeederPosition: LREAL;
	lrToolRightPosition: LREAL;
	lrSaveToolFeederPosition: LREAL;
	lrSaveToolRightPosition: LREAL;
	rPlungeCycleGrindFeedGeometry: REAL;
	lrGearFactor: LREAL;
	xPositionReached: BOOL;
	lrToolFeedCalcLengthPosition: REAL;
	lrCalcToolLengthInc: LREAL;
	lrCalcToolLength: LREAL;
	xReadyToolFeedStop: BOOL;
	xReadyGrindFeedStop: BOOL;
END_VAR
(****************************************************************************************************************************************************)
(***********                                This Functionblock define the function for work a geometry on the tool                                          ************)
(****************************************************************************************************************************************************)

